C07275=1014.277,-66.718,394.005,165.149,59.305,160.508
C07276=1014.282,-66.468,393.994,165.151,59.299,160.507
C07277=1014.287,-66.219,393.985,165.154,59.292,160.507
C07278=1014.291,-65.969,393.976,165.157,59.286,160.507
C07279=1014.296,-65.719,393.966,165.160,59.279,160.506
C07280=1014.301,-65.470,393.956,165.161,59.272,160.505
C07281=1014.306,-65.219,393.947,165.165,59.265,160.505
C07282=1014.311,-64.970,393.937,165.167,59.258,160.504
C07283=1014.316,-64.720,393.927,165.170,59.251,160.504
C07284=1014.320,-64.470,393.918,165.173,59.245,160.503
C07285=1014.325,-64.221,393.908,165.175,59.238,160.502
C07286=1014.331,-63.971,393.898,165.177,59.231,160.502
C07287=1014.335,-63.721,393.889,165.180,59.223,160.501
C07288=1014.340,-63.472,393.879,165.183,59.217,160.501
C07289=1014.345,-63.222,393.869,165.186,59.210,160.500
C07290=1014.350,-62.972,393.859,165.187,59.203,160.500
C07291=1014.355,-62.722,393.850,165.190,59.196,160.499
C07292=1014.360,-62.473,393.840,165.193,59.189,160.498
C07293=1014.364,-62.223,393.830,165.196,59.182,160.498
C07294=1014.370,-61.973,393.820,165.199,59.175,160.497
C07295=1014.374,-61.723,393.811,165.201,59.168,160.497
C07296=1014.379,-61.474,393.801,165.203,59.161,160.496
C07297=1014.384,-61.224,393.792,165.205,59.154,160.495
C07298=1014.390,-60.974,393.781,165.208,59.147,160.495
C07299=1014.394,-60.724,393.772,165.211,59.140,160.494
C07300=1014.399,-60.475,393.763,165.214,59.133,160.494
C07301=1014.404,-60.225,393.752,165.217,59.126,160.493
C07302=1014.409,-59.975,393.743,165.219,59.119,160.493
C07303=1014.413,-59.725,393.732,165.222,59.112,160.492
C07304=1014.418,-59.475,393.723,165.225,59.104,160.492
C07305=1014.423,-59.225,393.713,165.227,59.097,160.491
C07306=1014.428,-58.976,393.703,165.229,59.091,160.490
C07307=1014.433,-58.726,393.693,165.231,59.083,160.489
C07308=1014.438,-58.476,393.683,165.234,59.076,160.489
C07309=1014.443,-58.227,393.673,165.237,59.069,160.488
C07310=1014.449,-57.977,393.663,165.239,59.062,160.488
C07311=1014.453,-57.727,393.654,165.242,59.055,160.487
C07312=1014.458,-57.477,393.644,165.245,59.048,160.486
C07313=1014.463,-57.227,393.634,165.247,59.040,160.486
C07314=1014.468,-56.978,393.624,165.250,59.033,160.485
C07315=1014.474,-56.728,393.614,165.253,59.026,160.485
C07316=1014.478,-56.478,393.604,165.255,59.018,160.484
C07317=1014.483,-56.229,393.595,165.257,59.011,160.483
C07318=1014.489,-55.979,393.584,165.260,59.004,160.483
C07319=1014.494,-55.729,393.575,165.263,58.997,160.482
C07320=1014.498,-55.480,393.565,165.265,58.989,160.481
C07321=1014.504,-55.229,393.555,165.268,58.982,160.481
C07322=1014.508,-54.980,393.546,165.271,58.975,160.480
C07323=1014.514,-54.730,393.535,165.273,58.967,160.479
C07324=1014.519,-54.480,393.526,165.275,58.960,160.479
C07325=1014.524,-54.204,393.514,165.278,58.952,160.478
C07326=1014.530,-53.930,393.503,165.282,58.944,160.477
C07327=1014.535,-53.653,393.492,165.284,58.936,160.477
C07328=1014.541,-53.378,393.481,165.287,58.928,160.476
C07329=1014.546,-53.128,393.471,165.290,58.921,160.475
C07330=1014.551,-52.879,393.461,165.292,58.913,160.474
C07331=1014.556,-52.629,393.451,165.295,58.906,160.474
C07332=1014.561,-52.379,393.441,165.298,58.898,160.473
C07333=1014.566,-52.130,393.432,165.300,58.890,160.472
C07334=1014.572,-51.880,393.421,165.303,58.883,160.472
C07335=1014.576,-51.630,393.412,165.306,58.876,160.471
C07336=1014.581,-51.380,393.401,165.308,58.868,160.470
C07337=1014.586,-51.130,393.391,165.310,58.861,160.470
C07338=1014.591,-50.880,393.381,165.313,58.854,160.469
C07339=1014.596,-50.631,393.369,165.316,58.847,160.468
C07340=1014.601,-50.381,393.360,165.318,58.839,160.468
C07341=1014.606,-50.131,393.349,165.321,58.832,160.467
C07342=1014.611,-49.881,393.339,165.324,58.825,160.467
C07343=1014.616,-49.632,393.328,165.326,58.818,160.466
C07344=1014.621,-49.382,393.318,165.329,58.811,160.465
C07345=1014.625,-49.132,393.307,165.331,58.803,160.464
C07346=1014.630,-48.883,393.297,165.334,58.796,160.464
C07347=1014.636,-48.633,393.286,165.337,58.789,160.463
C07348=1014.640,-48.383,393.276,165.339,58.782,160.463
C07349=1014.646,-48.134,393.265,165.342,58.774,160.462
C07350=1014.650,-47.883,393.254,165.345,58.767,160.461
C07351=1014.655,-47.634,393.245,165.347,58.759,160.461
C07352=1014.660,-47.384,393.233,165.349,58.752,160.460
C07353=1014.665,-47.135,393.223,165.352,58.745,160.459
C07354=1014.670,-46.884,393.213,165.355,58.738,160.459
C07355=1014.675,-46.635,393.202,165.357,58.730,160.458
C07356=1014.680,-46.385,393.191,165.359,58.723,160.457
C07357=1014.685,-46.135,393.180,165.362,58.716,160.457
C07358=1014.689,-45.886,393.170,165.365,58.709,160.456
C07359=1014.695,-45.636,393.160,165.367,58.701,160.455
C07360=1014.699,-45.386,393.149,165.370,58.694,160.454
C07361=1014.705,-45.136,393.139,165.372,58.687,160.454
C07362=1014.710,-44.887,393.128,165.374,58.679,160.453
C07363=1014.714,-44.637,393.117,165.377,58.672,160.452
C07364=1014.720,-44.388,393.106,165.380,58.664,160.452
C07365=1014.725,-44.137,393.096,165.383,58.656,160.451
C07366=1014.730,-43.888,393.086,165.386,58.649,160.450
C07367=1014.735,-43.638,393.074,165.388,58.642,160.450
C07368=1014.740,-43.389,393.065,165.390,58.634,160.449
C07369=1014.745,-43.139,393.053,165.393,58.627,160.448
C07370=1014.750,-42.889,393.043,165.395,58.619,160.447
C07371=1014.754,-42.640,393.032,165.398,58.612,160.447
C07372=1014.760,-42.390,393.022,165.400,58.604,160.446
C07373=1014.765,-42.140,393.010,165.404,58.596,160.445
C07374=1014.770,-41.890,393.000,165.406,58.589,160.445
C07375=1014.775,-41.641,392.989,165.409,58.582,160.444
C07376=1014.780,-41.390,392.979,165.411,58.574,160.443
C07377=1014.785,-41.141,392.967,165.413,58.567,160.442
C07378=1014.790,-40.891,392.958,165.416,58.559,160.442
C07379=1014.795,-40.641,392.946,165.419,58.551,160.441
C07380=1014.800,-40.391,392.936,165.421,58.543,160.440
C07381=1014.806,-40.143,392.925,165.424,58.536,160.440
C07382=1014.811,-39.893,392.914,165.426,58.528,160.439
C07383=1014.816,-39.643,392.904,165.429,58.521,160.438
C07384=1014.821,-39.393,392.892,165.431,58.513,160.437
C07385=1014.825,-39.143,392.882,165.434,58.506,160.437
C07386=1014.830,-38.893,392.870,165.438,58.499,160.436
C07387=1014.836,-38.644,392.860,165.440,58.491,160.435
C07388=1014.840,-38.395,392.848,165.442,58.484,160.435
C07389=1014.846,-38.119,392.837,165.445,58.476,160.434
C07390=1014.852,-37.844,392.824,165.448,58.468,160.433
C07391=1014.857,-37.568,392.812,165.450,58.459,160.432
C07392=1014.862,-37.293,392.800,165.453,58.450,160.431
C07393=1014.867,-37.043,392.789,165.456,58.443,160.431
C07394=1014.872,-36.793,392.777,165.458,58.435,160.430
C07395=1014.877,-36.544,392.766,165.461,58.428,160.429
C07396=1014.882,-36.295,392.755,165.463,58.420,160.428
C07397=1014.887,-36.044,392.745,165.466,58.413,160.428
C07398=1014.892,-35.795,392.733,165.468,58.405,160.427
C07399=1014.897,-35.545,392.722,165.472,58.398,160.426
C07400=1014.902,-35.295,392.710,165.474,58.390,160.425
C07401=1014.907,-35.046,392.700,165.477,58.383,160.425
C07402=1014.912,-34.796,392.689,165.479,58.375,160.424
C07403=1014.917,-34.546,392.678,165.481,58.367,160.423
C07404=1014.922,-34.296,392.666,165.484,58.360,160.422
C07405=1014.928,-34.047,392.655,165.487,58.352,160.422
C07406=1014.932,-33.798,392.644,165.490,58.345,160.421
C07407=1014.937,-33.548,392.633,165.492,58.337,160.420
C07408=1014.942,-33.298,392.621,165.494,58.329,160.419
C07409=1014.948,-33.048,392.611,165.497,58.322,160.419
C07410=1014.953,-32.798,392.600,165.500,58.314,160.418
C07411=1014.958,-32.548,392.588,165.502,58.306,160.417
C07412=1014.963,-32.299,392.577,165.505,58.299,160.417
C07413=1014.967,-32.049,392.565,165.507,58.291,160.416
C07414=1014.973,-31.800,392.555,165.510,58.283,160.415
C07415=1014.978,-31.550,392.543,165.512,58.275,160.414
C07416=1014.983,-31.300,392.532,165.515,58.268,160.413
C07417=1014.988,-31.051,392.520,165.517,58.260,160.412
C07418=1014.994,-30.801,392.509,165.519,58.252,160.412
C07419=1014.998,-30.551,392.499,165.523,58.245,160.411
C07420=1015.003,-30.301,392.487,165.525,58.237,160.410
C07421=1015.008,-30.051,392.476,165.527,58.229,160.409
C07422=1015.013,-29.802,392.465,165.531,58.221,160.409
C07423=1015.018,-29.552,392.454,165.533,58.213,160.408
C07424=1015.023,-29.303,392.442,165.536,58.206,160.407
C07425=1015.028,-29.053,392.431,165.538,58.198,160.406
C07426=1015.033,-28.803,392.419,165.541,58.190,160.406
C07427=1015.039,-28.554,392.408,165.543,58.182,160.405
C07428=1015.044,-28.304,392.397,165.545,58.174,160.404
C07429=1015.049,-28.054,392.385,165.548,58.166,160.403
C07430=1015.054,-27.804,392.374,165.551,58.158,160.402
C07431=1015.059,-27.554,392.362,165.553,58.151,160.401
C07432=1015.064,-27.305,392.351,165.556,58.143,160.401
C07433=1015.069,-27.055,392.339,165.558,58.136,160.400
C07434=1015.074,-26.806,392.327,165.562,58.128,160.399
C07435=1015.079,-26.556,392.316,165.564,58.120,160.398
C07436=1015.084,-26.306,392.304,165.566,58.113,160.397
C07437=1015.089,-26.056,392.293,165.568,58.105,160.397
C07438=1015.095,-25.807,392.281,165.571,58.098,160.396
C07439=1015.100,-25.557,392.269,165.574,58.089,160.395
C07440=1015.105,-25.307,392.258,165.576,58.082,160.394
C07441=1015.110,-25.058,392.246,165.579,58.074,160.393
C07442=1015.115,-24.808,392.235,165.581,58.067,160.393
C07443=1015.120,-24.559,392.223,165.585,58.059,160.392
C07444=1015.124,-24.308,392.211,165.587,58.051,160.391
C07445=1015.129,-24.059,392.199,165.589,58.043,160.390
C07446=1015.134,-23.809,392.188,165.591,58.035,160.389
C07447=1015.140,-23.560,392.175,165.595,58.028,160.389
C07448=1015.145,-23.310,392.164,165.597,58.020,160.388
C07449=1015.150,-23.060,392.152,165.599,58.012,160.387
C07450=1015.155,-22.811,392.140,165.602,58.004,160.386
C07451=1015.160,-22.561,392.129,165.605,57.996,160.386
C07452=1015.165,-22.311,392.117,165.607,57.988,160.385
C07453=1015.171,-22.035,392.104,165.610,57.979,160.384
C07454=1015.176,-21.758,392.091,165.613,57.971,160.383
C07455=1015.182,-21.483,392.079,165.616,57.962,160.382
C07456=1015.188,-21.207,392.065,165.618,57.953,160.381
C07457=1015.193,-20.957,392.054,165.621,57.946,160.380
C07458=1015.198,-20.707,392.042,165.623,57.938,160.380
C07459=1015.204,-20.457,392.030,165.627,57.930,160.379
C07460=1015.208,-20.207,392.018,165.629,57.922,160.378
C07461=1015.213,-19.957,392.006,165.631,57.915,160.377
C07462=1015.218,-19.708,391.994,165.634,57.906,160.376
C07463=1015.223,-19.458,391.983,165.636,57.899,160.375
C07464=1015.228,-19.209,391.970,165.639,57.891,160.375
C07465=1015.233,-18.959,391.959,165.642,57.883,160.374
C07466=1015.238,-18.709,391.947,165.643,57.874,160.373
C07467=1015.244,-18.460,391.935,165.646,57.866,160.372
C07468=1015.249,-18.210,391.924,165.649,57.858,160.371
C07469=1015.255,-17.961,391.911,165.651,57.850,160.370
C07470=1015.260,-17.711,391.900,165.653,57.843,160.369
C07471=1015.265,-17.461,391.888,165.657,57.834,160.369
C07472=1015.270,-17.212,391.876,165.659,57.827,160.368
C07473=1015.275,-16.962,391.865,165.662,57.818,160.367
C07474=1015.280,-16.712,391.852,165.664,57.811,160.366
C07475=1015.285,-16.462,391.840,165.667,57.803,160.365
C07476=1015.290,-16.212,391.829,165.669,57.794,160.364
C07477=1015.295,-15.963,391.816,165.672,57.786,160.363
C07478=1015.301,-15.714,391.804,165.674,57.778,160.362
C07479=1015.305,-15.464,391.792,165.677,57.770,160.362
C07480=1015.311,-15.214,391.780,165.680,57.763,160.361
C07481=1015.316,-14.964,391.768,165.682,57.756,160.360
C07482=1015.320,-14.714,391.755,165.684,57.748,160.359
C07483=1015.326,-14.465,391.743,165.688,57.740,160.359
C07484=1015.330,-14.215,391.731,165.690,57.732,160.358
C07485=1015.336,-13.965,391.719,165.692,57.723,160.356
C07486=1015.341,-13.715,391.707,165.695,57.715,160.356
C07487=1015.346,-13.466,391.694,165.697,57.707,160.355
C07488=1015.351,-13.217,391.682,165.699,57.700,160.354
C07489=1015.356,-12.967,391.671,165.703,57.691,160.353
C07490=1015.361,-12.717,391.657,165.705,57.684,160.352
C07491=1015.366,-12.468,391.645,165.707,57.676,160.351
C07492=1015.372,-12.218,391.633,165.709,57.668,160.351
C07493=1015.376,-11.968,391.621,165.713,57.660,160.350
C07494=1015.382,-11.718,391.608,165.715,57.652,160.349
C07495=1015.387,-11.469,391.596,165.717,57.645,160.348
C07496=1015.391,-11.219,391.584,165.721,57.636,160.347
C07497=1015.397,-10.970,391.572,165.722,57.628,160.346
C07498=1015.403,-10.720,391.559,165.726,57.620,160.345
C07499=1015.407,-10.471,391.547,165.728,57.612,160.345
C07500=1015.412,-10.221,391.535,165.730,57.604,160.344
C07501=1015.417,-9.971,391.522,165.733,57.596,160.343
C07502=1015.423,-9.721,391.510,165.735,57.588,160.342
C07503=1015.428,-9.472,391.498,165.737,57.580,160.341
C07504=1015.432,-9.222,391.486,165.741,57.572,160.340
C07505=1015.438,-8.972,391.473,165.743,57.564,160.339
C07506=1015.443,-8.723,391.461,165.745,57.556,160.338
C07507=1015.448,-8.474,391.448,165.748,57.547,160.337
C07508=1015.453,-8.224,391.437,165.750,57.540,160.337
C07509=1015.460,-7.880,391.420,165.754,57.528,160.335
C07510=1015.468,-7.536,391.402,165.758,57.517,160.334
C07511=1015.475,-7.193,391.385,165.761,57.506,160.333
C07512=1015.482,-6.850,391.368,165.765,57.495,160.332
C07513=1015.486,-6.632,391.358,165.767,57.488,160.331
C07514=1015.491,-6.415,391.346,165.769,57.480,160.330
C07515=1015.496,-6.199,391.335,165.771,57.474,160.329
C07516=1015.500,-5.982,391.324,165.773,57.466,160.328
C07517=1015.505,-5.765,391.314,165.775,57.460,160.328
C07518=1015.509,-5.548,391.303,165.778,57.453,160.327
C07519=1015.514,-5.331,391.292,165.780,57.445,160.326
C07520=1015.518,-5.114,391.281,165.782,57.438,160.325
C07521=1015.523,-4.865,391.270,165.785,57.430,160.325
C07522=1015.528,-4.614,391.257,165.787,57.422,160.323
C07523=1015.534,-4.365,391.245,165.790,57.414,160.323
C07524=1015.539,-4.115,391.231,165.793,57.406,160.322
C07525=1015.543,-3.866,391.219,165.795,57.398,160.321
C07526=1015.548,-3.616,391.206,165.797,57.390,160.320
C07527=1015.554,-3.367,391.193,165.800,57.382,160.319
C07528=1015.559,-3.117,391.180,165.802,57.374,160.318
C07529=1015.564,-2.867,391.167,165.805,57.366,160.317
C07530=1015.568,-2.618,391.154,165.808,57.358,160.317
C07531=1015.574,-2.368,391.142,165.810,57.350,160.316
C07532=1015.579,-2.118,391.129,165.812,57.342,160.315
C07533=1015.583,-1.869,391.116,165.815,57.334,160.314
C07534=1015.589,-1.619,391.103,165.818,57.326,160.313
C07535=1015.594,-1.370,391.090,165.820,57.318,160.312
C07536=1015.599,-1.120,391.077,165.822,57.310,160.311
C07537=1015.604,-0.870,391.064,165.825,57.302,160.310
C07538=1015.609,-0.621,391.052,165.828,57.294,160.309
C07539=1015.614,-0.371,391.038,165.830,57.286,160.308
C07540=1015.619,-0.121,391.026,165.833,57.277,160.307
C07541=1015.624,0.129,391.013,165.835,57.270,160.307
C07542=1015.630,0.377,391.000,165.838,57.262,160.306
C07543=1015.635,0.628,390.986,165.840,57.253,160.305
C07544=1015.639,0.877,390.974,165.842,57.245,160.304
C07545=1015.644,1.127,390.961,165.846,57.237,160.303
C07546=1015.650,1.376,390.948,165.848,57.229,160.302
C07547=1015.655,1.625,390.935,165.850,57.221,160.301
C07548=1015.660,1.875,390.922,165.853,57.213,160.300
C07549=1015.665,2.125,390.909,165.855,57.205,160.299
C07550=1015.670,2.375,390.896,165.857,57.197,160.298
C07551=1015.675,2.624,390.883,165.861,57.189,160.298
C07552=1015.681,2.874,390.870,165.862,57.180,160.296
C07553=1015.685,3.123,390.857,165.866,57.172,160.296
C07554=1015.691,3.373,390.844,165.868,57.164,160.295
C07555=1015.696,3.622,390.831,165.870,57.156,160.294
C07556=1015.701,3.872,390.818,165.873,57.148,160.293
C07557=1015.706,4.122,390.805,165.875,57.140,160.292
C07558=1015.712,4.372,390.792,165.879,57.132,160.291
C07559=1015.716,4.621,390.779,165.880,57.123,160.290
C07560=1015.722,4.871,390.766,165.883,57.116,160.289
C07561=1015.726,5.120,390.753,165.886,57.107,160.288
C07562=1015.732,5.370,390.740,165.888,57.099,160.287
C07563=1015.738,5.620,390.727,165.891,57.090,160.286
C07564=1015.742,5.869,390.714,165.893,57.083,160.285
C07565=1015.748,6.119,390.700,165.896,57.074,160.284
C07566=1015.753,6.368,390.688,165.898,57.066,160.284
C07567=1015.758,6.618,390.675,165.901,57.057,160.283
C07568=1015.763,6.867,390.661,165.903,57.050,160.282
C07569=1015.768,7.117,390.648,165.905,57.041,160.280
C07570=1015.774,7.367,390.635,165.909,57.033,160.280
C07571=1015.779,7.616,390.622,165.910,57.025,160.279
C07572=1015.784,7.866,390.609,165.913,57.016,160.278
C07573=1015.789,8.116,390.596,165.916,57.008,160.277
C07574=1015.795,8.365,390.583,165.919,56.999,160.276
C07575=1015.799,8.614,390.570,165.921,56.992,160.275
C07576=1015.805,8.865,390.557,165.924,56.983,160.274
C07577=1015.810,9.114,390.543,165.926,56.974,160.273
C07578=1015.815,9.363,390.531,165.929,56.966,160.272
C07579=1015.821,9.613,390.517,165.931,56.958,160.271
C07580=1015.825,9.862,390.504,165.934,56.949,160.270
C07581=1015.832,10.143,390.489,165.936,56.940,160.269
C07582=1015.837,10.423,390.474,165.939,56.931,160.268
C07583=1015.843,10.704,390.459,165.943,56.922,160.267
C07584=1015.849,10.984,390.445,165.945,56.912,160.266
C07585=1015.855,11.233,390.431,165.947,56.904,160.264
C07586=1015.860,11.483,390.419,165.950,56.896,160.264
C07587=1015.865,11.732,390.405,165.952,56.887,160.263
C07588=1015.870,11.982,390.392,165.955,56.878,160.262
C07589=1015.876,12.231,390.379,165.958,56.870,160.261
C07590=1015.881,12.481,390.366,165.960,56.862,160.260
C07591=1015.887,12.731,390.352,165.963,56.853,160.259
C07592=1015.891,12.980,390.339,165.965,56.845,160.258
C07593=1015.897,13.230,390.325,165.968,56.836,160.257
C07594=1015.902,13.480,390.312,165.970,56.828,160.256
C07595=1015.907,13.730,390.298,165.972,56.820,160.255
C07596=1015.912,13.979,390.285,165.976,56.812,160.254
C07597=1015.917,14.229,390.271,165.977,56.804,160.253
C07598=1015.923,14.478,390.258,165.981,56.795,160.252
C07599=1015.927,14.728,390.245,165.983,56.787,160.251
C07600=1015.933,14.977,390.231,165.986,56.778,160.250
C07601=1015.938,15.227,390.217,165.988,56.771,160.249
C07602=1015.943,15.476,390.204,165.990,56.762,160.248
C07603=1015.948,15.726,390.190,165.993,56.754,160.247
C07604=1015.954,15.976,390.177,165.995,56.746,160.246
C07605=1015.959,16.225,390.163,165.998,56.737,160.245
C07606=1015.963,16.475,390.149,166.000,56.729,160.244
C07607=1015.969,16.724,390.135,166.003,56.721,160.243
C07608=1015.974,16.974,390.122,166.005,56.712,160.242
C07609=1015.979,17.224,390.109,166.008,56.704,160.241
C07610=1015.984,17.473,390.095,166.011,56.696,160.240
C07611=1015.990,17.723,390.081,166.012,56.688,160.239
C07612=1015.995,17.972,390.067,166.015,56.679,160.238
C07613=1016.000,18.222,390.054,166.018,56.671,160.237
C07614=1016.005,18.471,390.041,166.021,56.662,160.236
C07615=1016.011,18.721,390.027,166.023,56.654,160.235
C07616=1016.016,18.970,390.013,166.025,56.645,160.234
C07617=1016.022,19.220,389.999,166.028,56.638,160.233
C07618=1016.025,19.470,389.986,166.031,56.629,160.232
C07619=1016.031,19.719,389.972,166.033,56.621,160.232
C07620=1016.036,19.969,389.958,166.035,56.613,160.230
C07621=1016.042,20.219,389.944,166.038,56.604,160.229
C07622=1016.047,20.467,389.930,166.040,56.596,160.228
C07623=1016.051,20.717,389.916,166.043,56.588,160.228
C07624=1016.057,20.967,389.902,166.045,56.579,160.226
C07625=1016.062,21.216,389.888,166.048,56.571,160.225
C07626=1016.068,21.467,389.875,166.051,56.563,160.225
C07627=1016.072,21.716,389.861,166.054,56.554,160.224
C07628=1016.077,21.965,389.847,166.056,56.546,160.222
C07629=1016.083,22.215,389.833,166.057,56.538,160.221
C07630=1016.088,22.465,389.819,166.061,56.530,160.221
C07631=1016.094,22.714,389.806,166.063,56.521,160.219
C07632=1016.098,22.963,389.791,166.066,56.513,160.219
C07633=1016.103,23.213,389.778,166.068,56.504,160.217
C07634=1016.109,23.463,389.764,166.071,56.496,160.217
C07635=1016.114,23.712,389.750,166.073,56.488,160.216
C07636=1016.120,23.962,389.736,166.076,56.479,160.215
C07637=1016.124,24.212,389.722,166.078,56.471,160.213
C07638=1016.130,24.461,389.708,166.081,56.462,160.212
C07639=1016.135,24.710,389.694,166.083,56.454,160.212
C07640=1016.140,24.960,389.680,166.086,56.446,160.211
C07641=1016.145,25.209,389.666,166.088,56.437,160.210
C07642=1016.150,25.459,389.652,166.091,56.429,160.209
C07643=1016.156,25.709,389.638,166.093,56.420,160.207
C07644=1016.161,25.958,389.624,166.096,56.412,160.206
C07645=1016.167,26.240,389.609,166.099,56.403,160.205
C07646=1016.173,26.521,389.593,166.102,56.393,160.204
C07647=1016.179,26.803,389.577,166.105,56.383,160.203
C07648=1016.184,27.085,389.561,166.107,56.374,160.202
C07649=1016.189,27.335,389.547,166.109,56.366,160.201
C07650=1016.195,27.584,389.532,166.112,56.357,160.200
C07651=1016.200,27.834,389.518,166.115,56.349,160.199
C07652=1016.205,28.083,389.504,166.118,56.341,160.198
C07653=1016.210,28.333,389.490,166.120,56.332,160.197
C07654=1016.216,28.583,389.476,166.122,56.324,160.196
C07655=1016.220,28.832,389.462,166.125,56.316,160.195
C07656=1016.225,29.081,389.447,166.127,56.308,160.194
C07657=1016.230,29.331,389.433,166.130,56.299,160.193
C07658=1016.236,29.580,389.419,166.132,56.291,160.192
C07659=1016.241,29.830,389.405,166.135,56.282,160.191
C07660=1016.246,30.080,389.390,166.138,56.274,160.190
C07661=1016.252,30.329,389.376,166.140,56.266,160.189
C07662=1016.256,30.579,389.361,166.143,56.257,160.188
C07663=1016.262,30.828,389.348,166.144,56.249,160.187
C07664=1016.267,31.078,389.333,166.147,56.240,160.186
C07665=1016.272,31.327,389.319,166.149,56.232,160.185
C07666=1016.277,31.577,389.304,166.152,56.223,160.184
C07667=1016.283,31.827,389.290,166.155,56.216,160.183
C07668=1016.287,32.076,389.276,166.158,56.207,160.182
C07669=1016.293,32.325,389.261,166.160,56.199,160.181
C07670=1016.298,32.575,389.247,166.163,56.190,160.180
C07671=1016.303,32.825,389.233,166.165,56.182,160.179
C07672=1016.308,33.074,389.218,166.168,56.173,160.178
C07673=1016.314,33.324,389.204,166.170,56.165,160.177
C07674=1016.319,33.574,389.189,166.173,56.156,160.176
C07675=1016.324,33.823,389.175,166.175,56.148,160.174
C07676=1016.329,34.072,389.160,166.178,56.139,160.174
C07677=1016.335,34.322,389.146,166.180,56.131,160.172
C07678=1016.339,34.572,389.132,166.183,56.122,160.171
C07679=1016.345,34.821,389.117,166.185,56.115,160.171
C07680=1016.351,35.070,389.104,166.188,56.106,160.170
C07681=1016.355,35.320,389.089,166.190,56.098,160.169
C07682=1016.361,35.569,389.075,166.193,56.089,160.168
C07683=1016.366,35.819,389.060,166.195,56.081,160.166
C07684=1016.372,36.068,389.045,166.198,56.072,160.165
C07685=1016.376,36.318,389.031,166.200,56.064,160.164
C07686=1016.381,36.568,389.017,166.204,56.055,160.163
C07687=1016.387,36.817,389.002,166.206,56.047,160.162
C07688=1016.392,37.067,388.988,166.207,56.039,160.161
C07689=1016.397,37.316,388.972,166.211,56.030,160.160
C07690=1016.401,37.566,388.958,166.213,56.022,160.159
C07691=1016.407,37.815,388.943,166.216,56.013,160.158
C07692=1016.412,38.065,388.929,166.218,56.005,160.157
C07693=1016.417,38.314,388.914,166.221,55.997,160.156
C07694=1016.422,38.564,388.900,166.223,55.988,160.155
C07695=1016.427,38.813,388.885,166.225,55.980,160.154
C07696=1016.433,39.063,388.869,166.228,55.972,160.153
C07697=1016.438,39.313,388.855,166.230,55.963,160.152
C07698=1016.444,39.562,388.840,166.233,55.955,160.151
C07699=1016.448,39.812,388.826,166.235,55.946,160.150
C07700=1016.453,40.061,388.810,166.238,55.938,160.149
C07701=1016.458,40.311,388.796,166.240,55.929,160.148
C07702=1016.464,40.560,388.781,166.243,55.921,160.147
C07703=1016.469,40.809,388.766,166.246,55.912,160.146
C07704=1016.474,41.059,388.752,166.248,55.904,160.145
C07705=1016.480,41.308,388.737,166.251,55.896,160.144
C07706=1016.484,41.558,388.723,166.253,55.887,160.143
C07707=1016.490,41.808,388.707,166.256,55.879,160.142
C07708=1016.495,42.057,388.692,166.258,55.870,160.140
C07709=1016.501,42.338,388.676,166.261,55.861,160.139
C07710=1016.507,42.620,388.659,166.264,55.852,160.138
C07711=1016.512,42.902,388.642,166.267,55.843,160.137
C07712=1016.518,43.184,388.625,166.270,55.833,160.136
C07713=1016.523,43.434,388.609,166.273,55.825,160.135
C07714=1016.528,43.683,388.595,166.275,55.816,160.134
C07715=1016.533,43.933,388.580,166.277,55.808,160.133
C07716=1016.538,44.182,388.565,166.280,55.800,160.132
C07717=1016.543,44.431,388.549,166.282,55.792,160.131
C07718=1016.548,44.680,388.534,166.284,55.784,160.130
C07719=1016.554,44.930,388.519,166.287,55.775,160.129
C07720=1016.558,45.180,388.504,166.290,55.767,160.128
C07721=1016.563,45.430,388.489,166.293,55.758,160.127
C07722=1016.568,45.679,388.474,166.295,55.750,160.126
C07723=1016.574,45.928,388.459,166.297,55.742,160.125
C07724=1016.579,46.177,388.443,166.300,55.734,160.124
C07725=1016.583,46.428,388.427,166.302,55.726,160.123
C07726=1016.589,46.677,388.412,166.304,55.717,160.122
C07727=1016.593,46.927,388.398,166.308,55.709,160.121
C07728=1016.598,47.176,388.383,166.310,55.701,160.120
C07729=1016.603,47.425,388.367,166.313,55.692,160.119
C07730=1016.608,47.675,388.352,166.315,55.684,160.118
C07731=1016.614,47.925,388.337,166.318,55.675,160.117
C07732=1016.619,48.174,388.321,166.320,55.667,160.116
C07733=1016.624,48.423,388.306,166.322,55.659,160.114
C07734=1016.629,48.672,388.291,166.325,55.650,160.114
C07735=1016.635,48.922,388.276,166.327,55.642,160.112
C07736=1016.640,49.172,388.261,166.330,55.633,160.111
C07737=1016.645,49.422,388.246,166.332,55.625,160.110
C07738=1016.650,49.671,388.231,166.336,55.616,160.109
C07739=1016.655,49.920,388.216,166.338,55.608,160.108
C07740=1016.660,50.170,388.200,166.340,55.600,160.107
C07741=1016.665,50.419,388.185,166.343,55.591,160.106
C07742=1016.670,50.669,388.170,166.345,55.583,160.105
C07743=1016.675,50.918,388.155,166.348,55.574,160.104
C07744=1016.681,51.168,388.139,166.350,55.566,160.103
C07745=1016.686,51.417,388.124,166.353,55.558,160.102
C07746=1016.691,51.666,388.109,166.355,55.549,160.101
C07747=1016.696,51.916,388.093,166.359,55.541,160.100
C07748=1016.702,52.166,388.078,166.361,55.533,160.099
C07749=1016.707,52.415,388.063,166.363,55.523,160.098
C07750=1016.712,52.664,388.048,166.365,55.515,160.097
C07751=1016.718,52.914,388.032,166.369,55.506,160.096
C07752=1016.722,53.164,388.016,166.371,55.498,160.095
C07753=1016.727,53.413,388.001,166.373,55.490,160.094
C07754=1016.732,53.662,387.986,166.376,55.481,160.093
C07755=1016.738,53.912,387.970,166.378,55.473,160.091
C07756=1016.743,54.161,387.955,166.381,55.465,160.091
C07757=1016.748,54.411,387.940,166.383,55.456,160.089
C07758=1016.753,54.661,387.924,166.386,55.447,160.088
C07759=1016.758,54.910,387.909,166.388,55.439,160.087
C07760=1016.763,55.159,387.894,166.391,55.430,160.086
C07761=1016.769,55.409,387.879,166.393,55.422,160.085
C07762=1016.774,55.658,387.863,166.397,55.414,160.084
C07763=1016.779,55.908,387.848,166.399,55.404,160.083
C07764=1016.785,56.158,387.833,166.401,55.396,160.082
C07765=1016.790,56.406,387.817,166.404,55.388,160.081
C07766=1016.795,56.656,387.802,166.407,55.379,160.080
C07767=1016.801,56.906,387.786,166.410,55.371,160.079
C07768=1016.806,57.155,387.771,166.411,55.362,160.077
C07769=1016.811,57.404,387.756,166.415,55.353,160.077
C07770=1016.817,57.654,387.740,166.417,55.345,160.075
C07771=1016.822,57.903,387.725,166.420,55.337,160.075
C07772=1016.826,58.153,387.709,166.422,55.328,160.073
C07773=1016.833,58.434,387.692,166.425,55.318,160.072
C07774=1016.839,58.716,387.675,166.428,55.309,160.071
C07775=1016.845,58.998,387.657,166.431,55.299,160.070
C07776=1016.850,59.280,387.640,166.434,55.289,160.068
C07777=1016.856,59.529,387.624,166.436,55.281,160.067
C07778=1016.861,59.778,387.609,166.439,55.272,160.066
C07779=1016.866,60.028,387.593,166.442,55.263,160.065
C07780=1016.872,60.278,387.578,166.444,55.255,160.064
C07781=1016.877,60.527,387.563,166.447,55.246,160.063
C07782=1016.882,60.777,387.547,166.449,55.237,160.062
C07783=1016.887,61.026,387.531,166.452,55.229,160.061
C07784=1016.892,61.275,387.515,166.454,55.221,160.060
C07785=1016.898,61.525,387.500,166.457,55.211,160.059
C07786=1016.903,61.774,387.485,166.460,55.203,160.058
C07787=1016.909,62.024,387.469,166.462,55.195,160.057
C07788=1016.914,62.273,387.453,166.465,55.185,160.055
C07789=1016.920,62.523,387.438,166.467,55.177,160.054
C07790=1016.925,62.772,387.423,166.470,55.169,160.053
C07791=1016.930,63.022,387.406,166.472,55.160,160.052
C07792=1016.935,63.271,387.391,166.476,55.152,160.051
C07793=1016.941,63.521,387.375,166.477,55.143,160.050
C07794=1016.945,63.770,387.359,166.481,55.135,160.049
C07795=1016.950,64.019,387.343,166.483,55.126,160.048
C07796=1016.956,64.269,387.328,166.486,55.118,160.047
C07797=1016.961,64.518,387.311,166.488,55.110,160.046
C07798=1016.966,64.768,387.296,166.491,55.100,160.045
C07799=1016.971,65.017,387.279,166.493,55.092,160.044
C07800=1016.976,65.267,387.264,166.496,55.084,160.043
C07801=1016.982,65.516,387.248,166.498,55.076,160.042
C07802=1016.987,65.766,387.232,166.502,55.067,160.041
C07803=1016.992,66.015,387.217,166.503,55.058,160.039
C07804=1016.997,66.265,387.200,166.507,55.050,160.038
C07805=1017.002,66.514,387.185,166.509,55.042,160.037
C07806=1017.008,66.763,387.168,166.512,55.033,160.036
C07807=1017.012,67.013,387.153,166.514,55.025,160.035
C07808=1017.018,67.262,387.136,166.516,55.016,160.034
C07809=1017.023,67.512,387.121,166.519,55.008,160.033
C07810=1017.028,67.761,387.104,166.521,54.999,160.032
C07811=1017.033,68.011,387.088,166.525,54.991,160.031
C07812=1017.039,68.260,387.072,166.527,54.983,160.030
C07813=1017.043,68.509,387.056,166.530,54.973,160.029
C07814=1017.049,68.759,387.040,166.532,54.965,160.028
C07815=1017.054,69.008,387.024,166.535,54.957,160.027
C07816=1017.059,69.258,387.008,166.537,54.949,160.026
C07817=1017.064,69.507,386.992,166.541,54.940,160.025
C07818=1017.070,69.756,386.975,166.543,54.932,160.024
C07819=1017.074,70.006,386.960,166.546,54.923,160.022
C07820=1017.079,70.256,386.943,166.548,54.915,160.021
C07821=1017.085,70.504,386.927,166.550,54.907,160.020
C07822=1017.090,70.755,386.911,166.553,54.898,160.019
C07823=1017.095,71.003,386.895,166.555,54.890,160.018
C07824=1017.100,71.253,386.878,166.558,54.881,160.017
C07825=1017.104,71.502,386.862,166.560,54.873,160.016
C07826=1017.110,71.752,386.846,166.564,54.864,160.015
C07827=1017.116,72.001,386.829,166.566,54.856,160.014
C07828=1017.121,72.251,386.814,166.569,54.848,160.013
C07829=1017.126,72.500,386.797,166.571,54.839,160.012
C07830=1017.130,72.749,386.781,166.574,54.830,160.011
C07831=1017.136,72.999,386.765,166.576,54.822,160.010
C07832=1017.141,73.248,386.749,166.580,54.814,160.009
C07833=1017.147,73.498,386.732,166.582,54.805,160.007
C07834=1017.152,73.747,386.716,166.585,54.796,160.006
C07835=1017.156,73.997,386.700,166.587,54.788,160.005
C07836=1017.162,74.246,386.683,166.590,54.780,160.004
C07837=1017.168,74.528,386.665,166.593,54.770,160.003
C07838=1017.174,74.809,386.647,166.595,54.761,160.002
C07839=1017.179,75.091,386.628,166.599,54.751,160.001
C07840=1017.185,75.373,386.609,166.602,54.741,159.999
C07841=1017.190,75.622,386.593,166.604,54.733,159.998
C07842=1017.196,75.871,386.577,166.607,54.724,159.997
C07843=1017.201,76.122,386.560,166.609,54.716,159.996
C07844=1017.206,76.370,386.545,166.612,54.707,159.995
C07845=1017.211,76.620,386.528,166.614,54.699,159.994
C07846=1017.216,76.870,386.511,166.618,54.691,159.993
C07847=1017.221,77.119,386.494,166.620,54.683,159.992
C07848=1017.227,77.368,386.478,166.623,54.673,159.991
C07849=1017.232,77.618,386.461,166.625,54.665,159.990
C07850=1017.237,77.867,386.445,166.627,54.657,159.989
C07851=1017.242,78.116,386.428,166.631,54.649,159.988
C07852=1017.247,78.365,386.411,166.633,54.641,159.987
C07853=1017.252,78.615,386.395,166.636,54.632,159.986
C07854=1017.257,78.865,386.378,166.638,54.623,159.984
C07855=1017.262,79.113,386.361,166.641,54.615,159.983
C07856=1017.267,79.363,386.344,166.644,54.607,159.982
C07857=1017.272,79.613,386.328,166.646,54.599,159.981
C07858=1017.277,79.862,386.311,166.649,54.590,159.980
C07859=1017.283,80.111,386.295,166.651,54.581,159.979
C07860=1017.288,80.361,386.278,166.654,54.573,159.978
C07861=1017.292,80.610,386.261,166.657,54.565,159.977
C07862=1017.298,80.859,386.245,166.660,54.557,159.976
C07863=1017.303,81.109,386.228,166.662,54.548,159.975
C07864=1017.307,81.358,386.211,166.665,54.539,159.974
C07865=1017.313,81.608,386.194,166.667,54.531,159.973
C07866=1017.318,81.857,386.178,166.670,54.523,159.972
C07867=1017.323,82.107,386.161,166.673,54.515,159.971
C07868=1017.328,82.356,386.144,166.675,54.506,159.969
C07869=1017.333,82.606,386.127,166.678,54.497,159.969
C07870=1017.339,82.855,386.111,166.681,54.489,159.968
C07871=1017.343,83.104,386.095,166.684,54.481,159.967
C07872=1017.349,83.354,386.078,166.686,54.472,159.965
C07873=1017.354,83.603,386.061,166.689,54.464,159.964
C07874=1017.359,83.853,386.044,166.691,54.456,159.963
C07875=1017.364,84.101,386.027,166.695,54.447,159.962
C07876=1017.369,84.351,386.010,166.697,54.438,159.961
C07877=1017.374,84.601,385.993,166.700,54.430,159.960
C07878=1017.379,84.850,385.977,166.702,54.422,159.959
C07879=1017.384,85.099,385.960,166.705,54.413,159.958
C07880=1017.389,85.349,385.943,166.707,54.405,159.957
C07881=1017.395,85.598,385.926,166.711,54.396,159.956
C07882=1017.401,85.848,385.910,166.713,54.388,159.955
C07883=1017.406,86.096,385.893,166.716,54.379,159.954
C07884=1017.411,86.346,385.876,166.718,54.371,159.953
C07885=1017.416,86.595,385.859,166.721,54.362,159.951
C07886=1017.421,86.845,385.842,166.724,54.354,159.950
C07887=1017.426,87.094,385.826,166.727,54.346,159.949
C07888=1017.431,87.344,385.809,166.729,54.337,159.948
C07889=1017.436,87.593,385.791,166.732,54.328,159.947
C07890=1017.442,87.842,385.774,166.734,54.320,159.946
C07891=1017.447,88.092,385.758,166.737,54.311,159.945
C07892=1017.452,88.341,385.741,166.740,54.303,159.944
C07893=1017.457,88.591,385.724,166.743,54.294,159.943
C07894=1017.462,88.840,385.707,166.746,54.286,159.942
C07895=1017.467,89.089,385.690,166.748,54.278,159.941
C07896=1017.473,89.339,385.673,166.751,54.270,159.940
C07897=1017.478,89.588,385.655,166.754,54.260,159.938
C07898=1017.483,89.837,385.639,166.756,54.252,159.937
C07899=1017.487,90.087,385.621,166.759,54.244,159.937
C07900=1017.493,90.336,385.604,166.762,54.236,159.935
C07901=1017.499,90.618,385.585,166.765,54.227,159.934
C07902=1017.504,90.899,385.565,166.768,54.217,159.933
C07903=1017.510,91.182,385.546,166.771,54.208,159.932
C07904=1017.515,91.463,385.527,166.774,54.198,159.931
C07905=1017.521,91.712,385.509,166.777,54.189,159.930
C07906=1017.525,91.962,385.492,166.779,54.181,159.928
C07907=1017.531,92.211,385.474,166.783,54.173,159.928
C07908=1017.536,92.461,385.457,166.785,54.165,159.926
C07909=1017.542,92.710,385.440,166.788,54.156,159.925
C07910=1017.546,92.960,385.422,166.790,54.148,159.924
C07911=1017.551,93.209,385.406,166.793,54.140,159.923
C07912=1017.556,93.458,385.388,166.796,54.131,159.922
C07913=1017.562,93.707,385.371,166.798,54.123,159.921
C07914=1017.566,93.957,385.353,166.801,54.114,159.920
C07915=1017.572,94.207,385.336,166.804,54.106,159.919
C07916=1017.577,94.456,385.319,166.807,54.097,159.918
C07917=1017.582,94.705,385.302,166.809,54.089,159.917
C07918=1017.587,94.955,385.284,166.812,54.081,159.916
C07919=1017.592,95.204,385.267,166.814,54.072,159.915
C07920=1017.597,95.453,385.250,166.818,54.064,159.914
C07921=1017.602,95.702,385.233,166.820,54.056,159.913
C07922=1017.607,95.952,385.215,166.824,54.047,159.912
C07923=1017.612,96.201,385.198,166.826,54.039,159.910
C07924=1017.618,96.450,385.180,166.829,54.030,159.909
C07925=1017.623,96.699,385.163,166.831,54.022,159.908
C07926=1017.628,96.949,385.145,166.834,54.013,159.907
C07927=1017.633,97.198,385.128,166.837,54.005,159.906
C07928=1017.639,97.448,385.111,166.840,53.996,159.905
C07929=1017.644,97.697,385.093,166.842,53.988,159.904
C07930=1017.649,97.947,385.076,166.846,53.980,159.903
C07931=1017.654,98.195,385.059,166.847,53.971,159.902
C07932=1017.659,98.444,385.041,166.851,53.963,159.901
C07933=1017.664,98.694,385.024,166.854,53.954,159.900
C07934=1017.669,98.943,385.006,166.856,53.946,159.899
C07935=1017.674,99.193,384.989,166.860,53.937,159.898
C07936=1017.680,99.442,384.972,166.862,53.929,159.897
C07937=1017.685,99.691,384.953,166.865,53.921,159.896
C07938=1017.689,99.941,384.935,166.868,53.912,159.894
C07939=1017.695,100.190,384.918,166.870,53.904,159.893
C07940=1017.699,100.440,384.900,166.873,53.896,159.892
C07941=1017.705,100.689,384.883,166.876,53.888,159.891
C07942=1017.710,100.938,384.865,166.879,53.879,159.890
C07943=1017.715,101.188,384.848,166.881,53.871,159.889
C07944=1017.720,101.437,384.830,166.885,53.862,159.888
C07945=1017.725,101.686,384.812,166.887,53.855,159.887
C07946=1017.730,101.936,384.794,166.889,53.846,159.886
C07947=1017.735,102.185,384.776,166.893,53.838,159.885
C07948=1017.740,102.435,384.759,166.895,53.830,159.884
C07949=1017.745,102.684,384.741,166.899,53.821,159.883
C07950=1017.750,102.933,384.723,166.900,53.813,159.882
C07951=1017.755,103.182,384.705,166.904,53.804,159.881
C07952=1017.760,103.431,384.687,166.906,53.796,159.880
C07953=1017.765,103.681,384.669,166.910,53.788,159.879
C07954=1017.771,103.930,384.652,166.912,53.779,159.878
C07955=1017.775,104.180,384.634,166.915,53.771,159.877
C07956=1017.781,104.429,384.617,166.918,53.763,159.876
C07957=1017.786,104.678,384.598,166.921,53.754,159.874
C07958=1017.791,104.927,384.581,166.923,53.746,159.873
C07959=1017.796,105.177,384.563,166.927,53.738,159.873
C07960=1017.801,105.426,384.545,166.929,53.730,159.871
C07961=1017.806,105.675,384.527,166.932,53.721,159.870
C07962=1017.811,105.924,384.509,166.935,53.713,159.869
C07963=1017.816,106.174,384.492,166.938,53.704,159.868
C07964=1017.821,106.423,384.474,166.940,53.696,159.867
C07965=1017.827,106.705,384.453,166.944,53.686,159.866
C07966=1017.834,106.987,384.433,166.947,53.677,159.865
C07967=1017.839,107.269,384.413,166.950,53.668,159.864
C07968=1017.845,107.551,384.392,166.954,53.658,159.863
C07969=1017.850,107.800,384.375,166.956,53.649,159.861
C07970=1017.855,108.050,384.357,166.959,53.641,159.860
C07971=1017.860,108.299,384.338,166.961,53.633,159.859
C07972=1017.865,108.549,384.322,166.965,53.624,159.858
C07973=1017.870,108.798,384.303,166.968,53.616,159.857
C07974=1017.875,109.047,384.286,166.970,53.607,159.856
C07975=1017.880,109.296,384.268,166.974,53.599,159.855
C07976=1017.886,109.545,384.250,166.976,53.591,159.854
C07977=1017.891,109.795,384.231,166.979,53.582,159.853
C07978=1017.896,110.044,384.213,166.982,53.574,159.852
C07979=1017.901,110.293,384.194,166.985,53.566,159.851
C07980=1017.906,110.543,384.177,166.988,53.558,159.850
C07981=1017.911,110.792,384.159,166.991,53.549,159.849
C07982=1017.916,111.041,384.141,166.993,53.541,159.848
C07983=1017.921,111.291,384.122,166.997,53.533,159.847
C07984=1017.926,111.540,384.105,166.999,53.524,159.845
C07985=1017.932,111.790,384.086,167.003,53.516,159.845
C07986=1017.937,112.038,384.067,167.005,53.508,159.843
C07987=1017.942,112.288,384.049,167.009,53.499,159.843
C07988=1017.946,112.537,384.031,167.011,53.491,159.841
C07989=1017.951,112.786,384.013,167.013,53.483,159.840
C07990=1017.956,113.035,383.994,167.017,53.475,159.839
C07991=1017.961,113.285,383.976,167.019,53.467,159.838
C07992=1017.966,113.535,383.957,167.023,53.458,159.837
C07993=1017.971,113.784,383.939,167.025,53.451,159.836
C07994=1017.976,114.033,383.920,167.029,53.442,159.835
C07995=1017.981,114.282,383.902,167.031,53.434,159.834
C07996=1017.986,114.531,383.884,167.033,53.426,159.833
C07997=1017.991,114.780,383.865,167.037,53.417,159.832
C07998=1017.996,115.030,383.847,167.039,53.410,159.831
C07999=1018.001,115.279,383.828,167.043,53.401,159.830
C08000=1018.006,115.528,383.810,167.045,53.393,159.829
C08001=1018.011,115.778,383.791,167.049,53.384,159.828
C08002=1018.016,116.026,383.773,167.051,53.377,159.827
C08003=1018.021,116.276,383.754,167.055,53.368,159.826
C08004=1018.026,116.526,383.736,167.057,53.360,159.825
C08005=1018.031,116.774,383.717,167.061,53.352,159.824
C08006=1018.035,117.024,383.698,167.063,53.343,159.823
C08007=1018.040,117.273,383.679,167.066,53.335,159.822
C08008=1018.045,117.522,383.661,167.069,53.327,159.821
C08009=1018.051,117.772,383.643,167.072,53.319,159.820
C08010=1018.056,118.021,383.624,167.074,53.310,159.819
C08011=1018.060,118.270,383.606,167.078,53.302,159.818
C08012=1018.066,118.519,383.587,167.081,53.294,159.817
C08013=1018.071,118.769,383.568,167.084,53.286,159.816
C08014=1018.076,119.018,383.549,167.087,53.278,159.815
C08015=1018.081,119.267,383.531,167.090,53.269,159.814
C08016=1018.086,119.517,383.513,167.092,53.261,159.813
C08017=1018.091,119.766,383.494,167.096,53.253,159.812
C08018=1018.096,120.015,383.476,167.099,53.245,159.811
C08019=1018.101,120.264,383.457,167.102,53.236,159.810
C08020=1018.106,120.513,383.439,167.104,53.228,159.809
C08021=1018.112,120.763,383.419,167.108,53.220,159.808
C08022=1018.116,121.012,383.401,167.110,53.212,159.807
C08023=1018.121,121.261,383.382,167.113,53.203,159.805
C08024=1018.126,121.510,383.364,167.116,53.195,159.804
C08025=1018.132,121.760,383.345,167.120,53.187,159.804
C08026=1018.137,122.009,383.327,167.122,53.179,159.802
C08027=1018.141,122.258,383.307,167.125,53.170,159.801
C08028=1018.146,122.508,383.289,167.128,53.163,159.800
C08029=1018.152,122.789,383.268,167.132,53.153,159.799
C08030=1018.158,123.071,383.247,167.135,53.144,159.798
C08031=1018.163,123.353,383.226,167.139,53.134,159.797
C08032=1018.169,123.635,383.205,167.142,53.125,159.796
C08033=1018.175,123.885,383.185,167.145,53.116,159.795
C08034=1018.180,124.134,383.167,167.148,53.109,159.794
C08035=1018.185,124.383,383.148,167.151,53.100,159.792
C08036=1018.191,124.632,383.129,167.153,53.092,159.791
C08037=1018.195,124.882,383.111,167.157,53.084,159.791
C08038=1018.201,125.130,383.092,167.160,53.075,159.789
C08039=1018.206,125.380,383.073,167.163,53.067,159.788
C08040=1018.211,125.629,383.055,167.166,53.059,159.787
C08041=1018.215,125.878,383.035,167.169,53.050,159.786
C08042=1018.221,126.128,383.017,167.172,53.042,159.785
C08043=1018.226,126.377,382.998,167.176,53.034,159.784
C08044=1018.231,126.626,382.979,167.178,53.025,159.783
C08045=1018.236,126.876,382.960,167.182,53.017,159.782
C08046=1018.241,127.125,382.941,167.184,53.009,159.781
C08047=1018.247,127.375,382.923,167.187,53.000,159.780
C08048=1018.252,127.623,382.904,167.191,52.992,159.779
C08049=1018.257,127.872,382.885,167.194,52.984,159.778
C08050=1018.263,128.122,382.866,167.197,52.975,159.777
C08051=1018.267,128.371,382.848,167.200,52.967,159.776
C08052=1018.273,128.620,382.828,167.203,52.959,159.775
C08053=1018.278,128.869,382.810,167.206,52.950,159.774
C08054=1018.283,129.118,382.791,167.209,52.942,159.773
C08055=1018.289,129.368,382.772,167.212,52.933,159.772
C08056=1018.293,129.617,382.753,167.216,52.925,159.771
C08057=1018.299,129.866,382.733,167.218,52.917,159.770
C08058=1018.303,130.116,382.715,167.222,52.909,159.769
C08059=1018.308,130.365,382.695,167.224,52.901,159.768
C08060=1018.314,130.614,382.677,167.228,52.892,159.767
C08061=1018.318,130.864,382.657,167.230,52.885,159.766
C08062=1018.324,131.113,382.638,167.234,52.876,159.765
C08063=1018.329,131.361,382.619,167.238,52.868,159.764
C08064=1018.334,131.611,382.599,167.240,52.860,159.763
C08065=1018.339,131.860,382.580,167.243,52.852,159.762
C08066=1018.344,132.110,382.560,167.246,52.844,159.761
C08067=1018.349,132.358,382.542,167.250,52.836,159.760
C08068=1018.354,132.608,382.522,167.252,52.828,159.759
C08069=1018.359,132.857,382.503,167.255,52.819,159.758
C08070=1018.364,133.107,382.484,167.259,52.811,159.757
C08071=1018.368,133.356,382.465,167.262,52.803,159.756
C08072=1018.374,133.605,382.446,167.265,52.795,159.755
C08073=1018.379,133.854,382.426,167.268,52.786,159.754
C08074=1018.384,134.104,382.407,167.271,52.778,159.753
C08075=1018.389,134.352,382.388,167.274,52.770,159.752
C08076=1018.394,134.602,382.368,167.278,52.762,159.751
C08077=1018.399,134.851,382.349,167.281,52.754,159.750
C08078=1018.404,135.101,382.329,167.283,52.745,159.749
C08079=1018.410,135.349,382.310,167.287,52.737,159.748
C08080=1018.415,135.599,382.290,167.290,52.729,159.747
C08081=1018.420,135.847,382.271,167.293,52.721,159.746
C08082=1018.425,136.097,382.251,167.297,52.712,159.745
C08083=1018.430,136.346,382.232,167.299,52.705,159.744
C08084=1018.435,136.596,382.213,167.303,52.696,159.743
C08085=1018.440,136.844,382.194,167.306,52.689,159.742
C08086=1018.445,137.094,382.174,167.309,52.680,159.741
C08087=1018.450,137.343,382.155,167.313,52.672,159.740
C08088=1018.455,137.592,382.135,167.315,52.664,159.739
C08089=1018.460,137.841,382.116,167.319,52.656,159.738
C08090=1018.465,138.090,382.096,167.322,52.648,159.737
C08091=1018.470,138.339,382.077,167.325,52.640,159.736
C08092=1018.475,138.589,382.057,167.329,52.631,159.735
C08093=1018.481,138.870,382.035,167.332,52.622,159.733
C08094=1018.486,139.152,382.012,167.335,52.613,159.732
C08095=1018.493,139.434,381.990,167.339,52.604,159.731
C08096=1018.498,139.717,381.968,167.343,52.595,159.730
C08097=1018.503,139.965,381.948,167.346,52.586,159.729
C08098=1018.508,140.215,381.928,167.350,52.578,159.728
C08099=1018.513,140.463,381.909,167.352,52.570,159.727
C08100=1018.518,140.713,381.889,167.356,52.562,159.726
C08101=1018.523,140.962,381.869,167.359,52.554,159.725
C08102=1018.527,141.211,381.849,167.362,52.546,159.724
C08103=1018.533,141.461,381.830,167.366,52.538,159.723
C08104=1018.538,141.709,381.810,167.368,52.530,159.722
C08105=1018.543,141.959,381.790,167.372,52.522,159.721
C08106=1018.548,142.208,381.771,167.375,52.514,159.720
C08107=1018.553,142.457,381.751,167.378,52.506,159.719
C08108=1018.558,142.707,381.731,167.382,52.498,159.718
C08109=1018.563,142.955,381.712,167.385,52.490,159.717
C08110=1018.568,143.204,381.691,167.388,52.481,159.716
C08111=1018.573,143.454,381.672,167.392,52.473,159.715
C08112=1018.579,143.702,381.652,167.394,52.465,159.714
C08113=1018.584,143.952,381.632,167.398,52.457,159.713
C08114=1018.588,144.202,381.612,167.402,52.449,159.713
C08115=1018.593,144.450,381.592,167.404,52.440,159.711
C08116=1018.599,144.700,381.573,167.408,52.432,159.710
C08117=1018.604,144.949,381.552,167.411,52.425,159.709
C08118=1018.608,145.198,381.533,167.414,52.416,159.708
C08119=1018.614,145.447,381.514,167.418,52.408,159.708
C08120=1018.619,145.696,381.493,167.420,52.400,159.706
C08121=1018.624,145.945,381.474,167.424,52.392,159.705
C08122=1018.629,146.194,381.453,167.428,52.384,159.705
C08123=1018.634,146.444,381.432,167.430,52.376,159.703
C08124=1018.639,146.693,381.413,167.434,52.368,159.703
C08125=1018.645,146.941,381.393,167.438,52.360,159.702
C08126=1018.650,147.191,381.373,167.441,52.352,159.701
C08127=1018.655,147.440,381.353,167.444,52.344,159.700
C08128=1018.659,147.689,381.333,167.448,52.336,159.699
C08129=1018.667,148.078,381.301,167.453,52.323,159.697
C08130=1018.675,148.468,381.269,167.457,52.310,159.696
C08131=1018.683,148.857,381.238,167.464,52.298,159.694
C08132=1018.691,149.246,381.207,167.468,52.285,159.693
C08133=1018.696,149.495,381.187,167.472,52.277,159.692
C08134=1018.701,149.744,381.167,167.475,52.270,159.691
C08135=1018.706,149.993,381.146,167.479,52.262,159.690
C08136=1018.711,150.242,381.126,167.482,52.253,159.689
C08137=1018.716,150.492,381.106,167.485,52.246,159.688
C08138=1018.721,150.740,381.085,167.489,52.238,159.687
C08139=1018.726,150.990,381.066,167.492,52.229,159.686
C08140=1018.731,151.239,381.045,167.495,52.221,159.685
C08141=1018.736,151.488,381.025,167.499,52.213,159.684
C08142=1018.741,151.737,381.004,167.502,52.205,159.683
C08143=1018.746,151.986,380.984,167.505,52.197,159.682
C08144=1018.751,152.235,380.964,167.509,52.189,159.681
C08145=1018.756,152.484,380.943,167.513,52.181,159.680
C08146=1018.762,152.733,380.923,167.515,52.173,159.679
C08147=1018.767,152.983,380.903,167.519,52.165,159.678
C08148=1018.771,153.232,380.883,167.523,52.157,159.677
C08149=1018.776,153.481,380.862,167.526,52.150,159.676
C08150=1018.782,153.730,380.842,167.529,52.141,159.675
C08151=1018.786,153.979,380.821,167.533,52.133,159.674
C08152=1018.791,154.228,380.800,167.536,52.125,159.673
C08153=1018.799,154.619,380.769,167.542,52.113,159.672
C08154=1018.807,155.010,380.736,167.547,52.100,159.670
C08155=1018.815,155.401,380.704,167.553,52.088,159.669
C08156=1018.823,155.792,380.672,167.557,52.075,159.668
C08157=1018.828,156.042,380.651,167.561,52.067,159.667
C08158=1018.833,156.290,380.631,167.565,52.059,159.666
C08159=1018.838,156.539,380.610,167.569,52.051,159.665
C08160=1018.843,156.788,380.590,167.572,52.044,159.664
C08161=1018.848,157.037,380.569,167.575,52.035,159.663
C08162=1018.853,157.287,380.548,167.579,52.027,159.662
C08163=1018.858,157.536,380.528,167.582,52.019,159.661
C08164=1018.863,157.785,380.507,167.585,52.011,159.660
C08165=1018.869,158.034,380.486,167.589,52.003,159.659
C08166=1018.874,158.283,380.466,167.593,51.995,159.658
C08167=1018.879,158.532,380.446,167.596,51.987,159.657
C08168=1018.883,158.781,380.425,167.600,51.979,159.656
C08169=1018.888,159.030,380.404,167.603,51.971,159.655
C08170=1018.893,159.279,380.382,167.607,51.964,159.654
C08171=1018.898,159.528,380.362,167.610,51.956,159.654
C08172=1018.903,159.778,380.340,167.614,51.948,159.653
C08173=1018.908,160.027,380.320,167.617,51.940,159.652
C08174=1018.913,160.276,380.298,167.621,51.932,159.651
C08175=1018.918,160.525,380.277,167.624,51.925,159.650
C08176=1018.922,160.773,380.257,167.628,51.917,159.649
C08177=1018.927,161.023,380.236,167.632,51.909,159.648
C08178=1018.932,161.271,380.214,167.634,51.902,159.647
C08179=1018.937,161.521,380.193,167.638,51.894,159.646
C08180=1018.941,161.770,380.172,167.642,51.886,159.645
C08181=1018.947,162.019,380.151,167.645,51.878,159.644
C08182=1018.951,162.268,380.130,167.649,51.871,159.644
C08183=1018.956,162.518,380.108,167.653,51.863,159.643
C08184=1018.962,162.766,380.087,167.656,51.855,159.642
C08185=1018.966,163.016,380.066,167.660,51.847,159.641
C08186=1018.972,163.264,380.045,167.663,51.839,159.640
C08187=1018.976,163.514,380.024,167.666,51.831,159.639
C08188=1018.981,163.763,380.002,167.670,51.824,159.638
C08189=1018.986,164.011,379.981,167.674,51.816,159.637
C08190=1018.991,164.261,379.960,167.677,51.808,159.636
C08191=1018.996,164.509,379.939,167.681,51.800,159.635
C08192=1019.001,164.759,379.918,167.685,51.792,159.634
C08193=1019.005,165.008,379.896,167.688,51.785,159.633
C08194=1019.011,165.257,379.875,167.691,51.777,159.632
C08195=1019.015,165.506,379.854,167.696,51.769,159.632
C08196=1019.021,165.755,379.833,167.700,51.761,159.631
C08197=1019.025,166.004,379.812,167.702,51.754,159.630
C08198=1019.030,166.253,379.790,167.706,51.746,159.629
C08199=1019.036,166.502,379.769,167.710,51.738,159.628
C08200=1019.040,166.751,379.747,167.714,51.730,159.627
C08201=1019.045,167.000,379.726,167.717,51.722,159.626
C08202=1019.050,167.249,379.705,167.721,51.715,159.625
C08203=1019.055,167.498,379.684,167.725,51.707,159.625
C08204=1019.061,167.747,379.663,167.729,51.699,159.624
C08205=1019.065,167.996,379.641,167.732,51.691,159.623
C08206=1019.070,168.245,379.620,167.735,51.683,159.622
C08207=1019.075,168.494,379.599,167.739,51.675,159.621
C08208=1019.080,168.743,379.577,167.743,51.667,159.620
C08209=1019.085,168.992,379.557,167.746,51.660,159.619
C08210=1019.091,169.242,379.534,167.750,51.652,159.618
C08211=1019.095,169.491,379.513,167.754,51.644,159.617
C08212=1019.101,169.740,379.492,167.758,51.636,159.616
C08213=1019.106,169.988,379.470,167.762,51.628,159.616
C08214=1019.110,170.238,379.449,167.765,51.621,159.615
C08215=1019.116,170.486,379.428,167.769,51.613,159.614
C08216=1019.120,170.736,379.406,167.772,51.605,159.613
C08217=1019.126,171.017,379.382,167.777,51.596,159.612
C08218=1019.132,171.299,379.358,167.781,51.587,159.611
C08219=1019.138,171.580,379.333,167.785,51.579,159.610
C08220=1019.143,171.862,379.309,167.790,51.570,159.609
C08221=1019.148,172.111,379.288,167.794,51.562,159.608
C08222=1019.154,172.359,379.266,167.798,51.554,159.607
C08223=1019.158,172.609,379.245,167.801,51.546,159.606
C08224=1019.164,172.858,379.223,167.804,51.538,159.605
C08225=1019.169,173.107,379.202,167.808,51.531,159.604
C08226=1019.174,173.356,379.181,167.812,51.523,159.603
C08227=1019.179,173.605,379.159,167.816,51.515,159.602
C08228=1019.184,173.853,379.137,167.820,51.507,159.602
C08229=1019.190,174.103,379.115,167.824,51.499,159.601
C08230=1019.195,174.352,379.095,167.828,51.491,159.600
C08231=1019.200,174.601,379.073,167.831,51.484,159.599
C08232=1019.205,174.850,379.051,167.835,51.476,159.598
C08233=1019.211,175.099,379.029,167.839,51.468,159.597
C08234=1019.215,175.348,379.008,167.843,51.460,159.596
C08235=1019.220,175.597,378.986,167.846,51.452,159.595
C08236=1019.226,175.846,378.965,167.850,51.444,159.594
C08237=1019.231,176.095,378.943,167.855,51.437,159.594
C08238=1019.236,176.344,378.921,167.859,51.429,159.593
C08239=1019.241,176.593,378.900,167.862,51.421,159.592
C08240=1019.246,176.842,378.878,167.866,51.413,159.591
C08241=1019.251,177.091,378.856,167.870,51.405,159.590
C08242=1019.257,177.340,378.835,167.874,51.397,159.589
C08243=1019.262,177.589,378.813,167.877,51.390,159.588
C08244=1019.268,177.838,378.791,167.881,51.382,159.587
C08245=1019.273,178.087,378.770,167.885,51.374,159.586
C08246=1019.277,178.336,378.748,167.889,51.367,159.586
C08247=1019.283,178.585,378.727,167.893,51.359,159.585
C08248=1019.288,178.834,378.705,167.897,51.351,159.584
C08249=1019.293,179.083,378.683,167.901,51.343,159.583
C08250=1019.299,179.331,378.662,167.905,51.335,159.582
C08251=1019.304,179.581,378.640,167.909,51.327,159.581
C08252=1019.309,179.830,378.618,167.913,51.319,159.580
C08253=1019.315,180.079,378.596,167.917,51.311,159.579
C08254=1019.320,180.328,378.574,167.921,51.303,159.578
C08255=1019.325,180.577,378.552,167.924,51.295,159.577
C08256=1019.331,180.826,378.531,167.929,51.288,159.577
C08257=1019.336,181.075,378.509,167.933,51.280,159.576
C08258=1019.341,181.323,378.487,167.937,51.272,159.575
C08259=1019.347,181.573,378.465,167.941,51.264,159.574
C08260=1019.352,181.821,378.444,167.945,51.256,159.573
C08261=1019.357,182.071,378.421,167.948,51.249,159.572
C08262=1019.362,182.320,378.399,167.953,51.241,159.572
C08263=1019.367,182.569,378.377,167.957,51.233,159.571
C08264=1019.372,182.818,378.354,167.961,51.226,159.570
C08265=1019.376,183.067,378.332,167.965,51.218,159.569
C08266=1019.382,183.316,378.310,167.969,51.210,159.568
C08267=1019.386,183.565,378.287,167.972,51.204,159.567
C08268=1019.392,183.814,378.265,167.976,51.196,159.566
C08269=1019.396,184.063,378.243,167.981,51.189,159.566
C08270=1019.401,184.312,378.219,167.984,51.181,159.565
C08271=1019.406,184.561,378.197,167.989,51.173,159.564
C08272=1019.411,184.809,378.175,167.993,51.166,159.563
C08273=1019.416,185.058,378.153,167.997,51.158,159.562
C08274=1019.421,185.308,378.130,168.001,51.150,159.562
C08275=1019.426,185.556,378.107,168.004,51.143,159.561
C08276=1019.431,185.806,378.085,168.008,51.136,159.560
C08277=1019.436,186.054,378.062,168.012,51.128,159.559
C08278=1019.441,186.304,378.040,168.017,51.121,159.558
C08279=1019.446,186.552,378.017,168.021,51.113,159.557
C08280=1019.451,186.802,377.994,168.025,51.105,159.556
C08281=1019.457,187.082,377.969,168.030,51.097,159.556
C08282=1019.462,187.363,377.944,168.034,51.088,159.555
C08283=1019.468,187.644,377.918,168.039,51.080,159.554
C08284=1019.474,187.925,377.893,168.043,51.071,159.553
C08285=1019.479,188.174,377.870,168.047,51.064,159.552
C08286=1019.484,188.423,377.847,168.051,51.056,159.551
C08287=1019.489,188.672,377.825,168.055,51.049,159.550
C08288=1019.494,188.921,377.802,168.059,51.041,159.550
C08289=1019.499,189.170,377.780,168.063,51.033,159.549
C08290=1019.505,189.419,377.757,168.068,51.026,159.548
C08291=1019.509,189.668,377.735,168.072,51.018,159.547
C08292=1019.514,189.917,377.712,168.076,51.011,159.546
C08293=1019.520,190.165,377.689,168.080,51.003,159.545
C08294=1019.525,190.415,377.667,168.084,50.996,159.545
C08295=1019.530,190.664,377.643,168.088,50.988,159.544
C08296=1019.535,190.912,377.621,168.093,50.981,159.543
C08297=1019.541,191.162,377.598,168.097,50.973,159.542
C08298=1019.545,191.410,377.575,168.101,50.965,159.541
C08299=1019.550,191.660,377.553,168.105,50.958,159.541
C08300=1019.556,191.908,377.530,168.109,50.950,159.540
C08301=1019.561,192.157,377.507,168.113,50.943,159.539
C08302=1019.566,192.406,377.484,168.118,50.935,159.538
C08303=1019.571,192.655,377.462,168.123,50.928,159.537
C08304=1019.576,192.904,377.439,168.127,50.920,159.537
C08305=1019.581,193.152,377.416,168.131,50.913,159.536
C08306=1019.587,193.402,377.394,168.135,50.905,159.535
C08307=1019.592,193.651,377.370,168.140,50.898,159.534
C08308=1019.597,193.899,377.348,168.144,50.890,159.533
C08309=1019.602,194.148,377.325,168.148,50.882,159.532
C08310=1019.607,194.398,377.302,168.152,50.875,159.532
C08311=1019.612,194.646,377.279,168.156,50.867,159.531
C08312=1019.618,194.895,377.256,168.160,50.860,159.530
C08313=1019.623,195.144,377.233,168.164,50.852,159.529
C08314=1019.628,195.392,377.210,168.169,50.845,159.528
C08315=1019.634,195.642,377.188,168.174,50.837,159.528
C08316=1019.639,195.891,377.164,168.178,50.830,159.527
C08317=1019.644,196.140,377.141,168.182,50.822,159.526
C08318=1019.649,196.388,377.119,168.186,50.815,159.525
C08319=1019.654,196.637,377.095,168.190,50.807,159.524
C08320=1019.660,196.886,377.072,168.195,50.800,159.524
C08321=1019.665,197.134,377.050,168.199,50.792,159.523
C08322=1019.670,197.384,377.026,168.204,50.784,159.522
C08323=1019.676,197.633,377.004,168.208,50.777,159.521
C08324=1019.681,197.882,376.981,168.212,50.769,159.520
C08325=1019.686,198.131,376.958,168.217,50.762,159.520
C08326=1019.692,198.379,376.935,168.221,50.754,159.519
C08327=1019.697,198.628,376.912,168.225,50.747,159.518
C08328=1019.702,198.878,376.888,168.230,50.739,159.517
C08329=1019.708,199.126,376.866,168.235,50.731,159.517
C08330=1019.713,199.375,376.843,168.239,50.724,159.516
C08331=1019.718,199.624,376.819,168.243,50.717,159.515
C08332=1019.723,199.873,376.796,168.247,50.709,159.514
C08333=1019.729,200.122,376.773,168.251,50.702,159.513
C08334=1019.734,200.371,376.749,168.256,50.695,159.513
C08335=1019.739,200.619,376.726,168.260,50.687,159.512
C08336=1019.744,200.868,376.703,168.265,50.679,159.511
C08337=1019.749,201.117,376.679,168.270,50.672,159.510
C08338=1019.755,201.366,376.655,168.274,50.665,159.510
C08339=1019.760,201.615,376.631,168.278,50.657,159.509
C08340=1019.765,201.863,376.609,168.283,50.650,159.508
C08341=1019.770,202.112,376.585,168.287,50.643,159.507
C08342=1019.775,202.361,376.561,168.291,50.635,159.506
C08343=1019.781,202.610,376.538,168.297,50.628,159.506
C08344=1019.786,202.859,376.514,168.301,50.621,159.505
C08345=1019.807,203.899,376.416,168.755,50.715,159.604
C08346=1019.812,204.119,376.394,168.758,50.709,159.603
C08347=1019.818,204.340,376.371,168.762,50.703,159.602
C08348=1019.824,204.561,376.349,168.765,50.698,159.602
C08349=1019.829,204.781,376.327,168.768,50.692,159.601
C08350=1019.835,205.003,376.305,168.771,50.686,159.600
C08351=1019.841,205.224,376.282,168.775,50.680,159.600
C08352=1019.846,205.444,376.260,168.778,50.675,159.599
C08353=1019.851,205.665,376.238,168.781,50.669,159.598
C08354=1019.857,205.914,376.213,168.784,50.663,159.598
C08355=1019.864,206.163,376.187,168.789,50.656,159.597
C08356=1019.869,206.412,376.161,168.793,50.650,159.596
C08357=1019.875,206.660,376.136,168.796,50.644,159.595
C08358=1019.881,206.908,376.111,168.800,50.637,159.595
C08359=1019.887,207.157,376.086,168.803,50.631,159.594
C08360=1019.893,207.406,376.060,168.807,50.625,159.593
C08361=1019.900,207.654,376.035,168.810,50.619,159.593
C08362=1019.906,207.903,376.010,168.814,50.613,159.592
C08363=1019.912,208.152,375.984,168.818,50.606,159.591
C08364=1019.918,208.400,375.959,168.821,50.600,159.590
C08365=1019.924,208.649,375.934,168.825,50.594,159.590
C08366=1019.931,208.898,375.908,168.829,50.588,159.589
C08367=1019.937,209.146,375.883,168.833,50.582,159.589
C08368=1019.943,209.395,375.858,168.836,50.575,159.588
C08369=1019.948,209.644,375.832,168.840,50.569,159.587
C08370=1019.955,209.893,375.806,168.843,50.563,159.586
C08371=1019.961,210.141,375.781,168.847,50.557,159.586
C08372=1019.966,210.389,375.756,168.851,50.551,159.585
C08373=1019.973,210.638,375.731,168.855,50.545,159.584
C08374=1019.978,210.886,375.704,168.858,50.538,159.584
C08375=1019.985,211.135,375.679,168.862,50.532,159.583
C08376=1019.991,211.384,375.653,168.866,50.526,159.582
C08377=1019.996,211.633,375.628,168.869,50.520,159.582
C08378=1020.003,211.881,375.602,168.873,50.514,159.581
C08379=1020.009,212.129,375.576,168.877,50.508,159.580
C08380=1020.015,212.378,375.550,168.881,50.502,159.580
C08381=1020.021,212.627,375.525,168.884,50.496,159.579
C08382=1020.027,212.876,375.500,168.888,50.490,159.578
C08383=1020.033,213.124,375.473,168.892,50.484,159.578
C08384=1020.039,213.373,375.448,168.895,50.478,159.577
C08385=1020.045,213.621,375.422,168.898,50.472,159.576
C08386=1020.052,213.869,375.396,168.902,50.466,159.576
C08387=1020.057,214.118,375.370,168.906,50.460,159.575
C08388=1020.064,214.368,375.344,168.910,50.454,159.574
C08389=1020.070,214.616,375.318,168.914,50.448,159.574
C08390=1020.076,214.865,375.293,168.917,50.442,159.573
C08391=1020.082,215.113,375.267,168.921,50.436,159.572
C08392=1020.089,215.361,375.241,168.925,50.430,159.572
C08393=1020.095,215.610,375.216,168.929,50.424,159.571
C08394=1020.100,215.859,375.190,168.932,50.417,159.570
C08395=1020.107,216.107,375.164,168.937,50.412,159.570
C08396=1020.113,216.356,375.138,168.940,50.406,159.569
C08397=1020.118,216.605,375.113,168.944,50.400,159.569
C08398=1020.125,216.853,375.086,168.948,50.394,159.568
C08399=1020.132,217.102,375.061,168.952,50.388,159.567
C08400=1020.138,217.351,375.034,168.955,50.382,159.567
C08401=1020.144,217.599,375.009,168.959,50.376,159.566
C08402=1020.150,217.847,374.983,168.962,50.370,159.565
C08403=1020.156,218.096,374.957,168.966,50.365,159.565
C08404=1020.162,218.344,374.931,168.970,50.359,159.564
C08405=1020.168,218.593,374.905,168.974,50.353,159.563
C08406=1020.177,218.962,374.867,168.980,50.345,159.563
C08407=1020.186,219.331,374.828,168.985,50.336,159.562
C08408=1020.195,219.700,374.789,168.990,50.328,159.561
C08409=1020.205,220.068,374.749,168.996,50.319,159.560
C08410=1020.210,220.317,374.723,169.000,50.313,159.559
C08411=1020.216,220.566,374.697,169.004,50.307,159.559
C08412=1020.222,220.814,374.671,169.008,50.302,159.558
C08413=1020.228,221.063,374.645,169.011,50.296,159.557
C08414=1020.235,221.312,374.618,169.015,50.291,159.557
C08415=1020.241,221.560,374.592,169.019,50.285,159.556
C08416=1020.246,221.809,374.566,169.023,50.279,159.556
C08417=1020.253,222.057,374.540,169.027,50.273,159.555
C08418=1020.258,222.305,374.513,169.031,50.267,159.555
C08419=1020.265,222.555,374.487,169.035,50.262,159.554
C08420=1020.271,222.803,374.461,169.038,50.256,159.553
C08421=1020.277,223.051,374.434,169.042,50.251,159.553
C08422=1020.283,223.299,374.408,169.046,50.245,159.552
C08423=1020.290,223.548,374.381,169.050,50.240,159.552
C08424=1020.296,223.797,374.356,169.054,50.234,159.551
C08425=1020.302,224.045,374.329,169.058,50.228,159.551
C08426=1020.307,224.294,374.302,169.061,50.223,159.550
C08427=1020.315,224.543,374.276,169.065,50.217,159.550
C08428=1020.320,224.791,374.249,169.069,50.211,159.549
C08429=1020.326,225.040,374.223,169.073,50.206,159.548
C08430=1020.332,225.288,374.197,169.077,50.200,159.548
C08431=1020.339,225.537,374.170,169.081,50.195,159.547
C08432=1020.345,225.785,374.144,169.084,50.189,159.547
C08433=1020.351,226.033,374.118,169.088,50.184,159.546
C08434=1020.357,226.283,374.091,169.091,50.178,159.545
C08435=1020.364,226.531,374.064,169.096,50.173,159.545
C08436=1020.370,226.779,374.038,169.100,50.167,159.544
C08437=1020.375,227.027,374.011,169.104,50.161,159.544
C08438=1020.382,227.276,373.984,169.107,50.156,159.543
C08439=1020.388,227.524,373.958,169.111,50.151,159.543
C08440=1020.394,227.773,373.931,169.115,50.146,159.542
C08441=1020.400,228.022,373.904,169.119,50.140,159.542
C08442=1020.406,228.270,373.878,169.123,50.134,159.541
C08443=1020.412,228.519,373.851,169.126,50.129,159.541
C08444=1020.418,228.768,373.824,169.131,50.124,159.540
C08445=1020.424,229.016,373.797,169.134,50.118,159.540
C08446=1020.432,229.342,373.762,169.139,50.112,159.539
C08447=1020.441,229.670,373.727,169.145,50.104,159.538
C08448=1020.449,229.996,373.692,169.150,50.097,159.538
C08449=1020.457,230.322,373.657,169.155,50.090,159.537
C08450=1020.463,230.571,373.630,169.159,50.085,159.536
C08451=1020.469,230.820,373.603,169.163,50.080,159.536
C08452=1020.475,231.067,373.576,169.166,50.075,159.535
C08453=1020.481,231.317,373.549,169.170,50.069,159.535
C08454=1020.487,231.565,373.522,169.174,50.064,159.534
C08455=1020.493,231.813,373.495,169.179,50.059,159.534
C08456=1020.500,232.062,373.468,169.182,50.054,159.533
C08457=1020.505,232.310,373.441,169.186,50.048,159.533
C08458=1020.512,232.559,373.414,169.190,50.043,159.533
C08459=1020.518,232.807,373.387,169.194,50.038,159.532
C08460=1020.524,233.056,373.360,169.198,50.033,159.532
C08461=1020.530,233.304,373.333,169.202,50.028,159.531
C08462=1020.535,233.524,373.309,169.205,50.023,159.531
C08463=1020.540,233.743,373.285,169.209,50.018,159.530
C08464=1020.546,233.963,373.261,169.212,50.014,159.530
C08465=1020.551,234.183,373.237,169.215,50.009,159.529
C08466=1020.557,234.402,373.213,169.219,50.005,159.529
C08467=1020.562,234.621,373.189,169.223,49.999,159.528
C08468=1020.568,234.841,373.165,169.227,49.995,159.528
C08469=1020.573,235.060,373.141,169.230,49.991,159.528
C08470=1020.579,235.309,373.114,169.233,49.986,159.527
C08471=1020.586,235.557,373.086,169.238,49.981,159.527
C08472=1020.591,235.805,373.060,169.242,49.975,159.526
C08473=1020.598,236.054,373.033,169.246,49.970,159.526
C08474=1020.604,236.302,373.005,169.249,49.965,159.525
C08475=1020.610,236.551,372.978,169.253,49.960,159.525
C08476=1020.617,236.800,372.951,169.258,49.954,159.524
C08477=1020.623,237.048,372.924,169.261,49.950,159.524
C08478=1020.629,237.296,372.896,169.265,49.945,159.524
C08479=1020.635,237.545,372.870,169.270,49.940,159.523
C08480=1020.641,237.794,372.841,169.274,49.934,159.523
C08481=1020.647,238.042,372.815,169.277,49.929,159.522
C08482=1020.653,238.290,372.787,169.281,49.925,159.522
C08483=1020.660,238.538,372.760,169.286,49.919,159.521
C08484=1020.666,238.787,372.732,169.290,49.914,159.521
C08485=1020.673,239.036,372.705,169.293,49.909,159.520
C08486=1020.678,239.284,372.678,169.298,49.905,159.520
C08487=1020.685,239.532,372.650,169.302,49.899,159.520
C08488=1020.690,239.780,372.622,169.305,49.894,159.519
C08489=1020.697,240.029,372.595,169.310,49.890,159.519
C08490=1020.702,240.278,372.567,169.314,49.885,159.518
C08491=1020.709,240.526,372.540,169.317,49.880,159.518
C08492=1020.715,240.774,372.512,169.322,49.875,159.517
C08493=1020.721,241.022,372.484,169.326,49.870,159.517
C08494=1020.727,241.272,372.457,169.329,49.865,159.517
C08495=1020.733,241.519,372.430,169.334,49.860,159.516
C08496=1020.739,241.768,372.401,169.338,49.856,159.516
C08497=1020.746,242.016,372.374,169.341,49.851,159.515
C08498=1020.751,242.265,372.346,169.346,49.846,159.515
C08499=1020.758,242.513,372.318,169.350,49.841,159.515
C08500=1020.764,242.762,372.291,169.354,49.836,159.514
C08501=1020.770,243.010,372.263,169.358,49.831,159.514
C08502=1020.776,243.259,372.235,169.363,49.827,159.514
C08503=1020.782,243.506,372.208,169.366,49.822,159.513
C08504=1020.788,243.755,372.180,169.370,49.817,159.513
C08505=1020.794,244.004,372.151,169.374,49.812,159.512
C08506=1020.800,244.251,372.124,169.378,49.808,159.512
C08507=1020.806,244.500,372.096,169.383,49.803,159.512
C08508=1020.812,244.749,372.067,169.386,49.798,159.511
C08509=1020.818,244.997,372.040,169.391,49.793,159.511
C08510=1020.825,245.245,372.011,169.394,49.789,159.510
C08511=1020.830,245.494,371.982,169.398,49.784,159.510
C08512=1020.837,245.741,371.955,169.403,49.779,159.510
C08513=1020.843,245.990,371.927,169.407,49.775,159.509
C08514=1020.848,246.239,371.898,169.411,49.770,159.509
C08515=1020.855,246.487,371.871,169.414,49.766,159.508
C08516=1020.860,246.735,371.843,169.419,49.761,159.508
C08517=1020.866,246.984,371.814,169.423,49.756,159.508
C08518=1020.873,247.232,371.786,169.427,49.752,159.508
C08519=1020.879,247.480,371.758,169.431,49.747,159.507
C08520=1020.885,247.729,371.730,169.435,49.743,159.507
C08521=1020.891,247.977,371.702,169.439,49.738,159.507
C08522=1020.897,248.193,371.677,169.443,49.734,159.506
C08523=1020.902,248.410,371.653,169.447,49.730,159.506
C08524=1020.907,248.625,371.628,169.451,49.726,159.506
C08525=1020.912,248.842,371.604,169.454,49.722,159.505
C08526=1020.918,249.059,371.579,169.457,49.718,159.505
C08527=1020.923,249.275,371.554,169.461,49.714,159.505
C08528=1020.929,249.491,371.529,169.465,49.710,159.505
C08529=1020.934,249.707,371.505,169.468,49.706,159.504
C08530=1020.940,249.956,371.476,169.473,49.702,159.504
C08531=1020.947,250.204,371.449,169.476,49.697,159.504
C08532=1020.953,250.453,371.420,169.481,49.693,159.503
C08533=1020.958,250.701,371.392,169.485,49.688,159.503
C08534=1020.965,250.949,371.364,169.489,49.683,159.502
C08535=1020.971,251.197,371.335,169.493,49.679,159.502
C08536=1020.977,251.446,371.307,169.497,49.674,159.502
C08537=1020.984,251.694,371.279,169.502,49.670,159.501
C08538=1020.990,251.943,371.250,169.506,49.665,159.501
C08539=1020.996,252.191,371.221,169.510,49.661,159.501
C08540=1021.002,252.439,371.194,169.514,49.656,159.501
C08541=1021.008,252.687,371.166,169.518,49.652,159.500
C08542=1021.014,252.935,371.137,169.523,49.648,159.500
C08543=1021.021,253.184,371.109,169.527,49.643,159.500
C08544=1021.027,253.432,371.080,169.531,49.639,159.499
C08545=1021.033,253.681,371.052,169.535,49.634,159.499
C08546=1021.040,253.929,371.023,169.540,49.630,159.499
C08547=1021.046,254.177,370.995,169.543,49.625,159.498
C08548=1021.052,254.425,370.966,169.548,49.621,159.498
C08549=1021.059,254.674,370.938,169.552,49.617,159.498
C08550=1021.065,254.922,370.909,169.556,49.612,159.497
C08551=1021.071,255.171,370.881,169.561,49.607,159.497
C08552=1021.078,255.419,370.852,169.564,49.603,159.497
C08553=1021.084,255.667,370.824,169.569,49.599,159.497
C08554=1021.090,255.916,370.795,169.574,49.594,159.496
C08555=1021.096,256.164,370.766,169.577,49.590,159.496
C08556=1021.103,256.412,370.738,169.582,49.586,159.496
C08557=1021.110,256.660,370.709,169.586,49.582,159.495
C08558=1021.115,256.909,370.681,169.590,49.577,159.495
C08559=1021.122,257.157,370.652,169.595,49.573,159.495
C08560=1021.128,257.406,370.624,169.599,49.568,159.495
C08561=1021.135,257.654,370.595,169.603,49.564,159.494
C08562=1021.142,257.902,370.566,169.608,49.559,159.494
C08563=1021.148,258.150,370.538,169.612,49.556,159.494
C08564=1021.154,258.398,370.509,169.616,49.551,159.494
C08565=1021.161,258.646,370.481,169.621,49.547,159.493
C08566=1021.167,258.895,370.452,169.625,49.542,159.493
C08567=1021.173,259.143,370.423,169.629,49.538,159.493
C08568=1021.180,259.391,370.395,169.633,49.534,159.492
C08569=1021.186,259.639,370.366,169.638,49.530,159.492
C08570=1021.192,259.888,370.337,169.642,49.525,159.492
C08571=1021.198,260.136,370.308,169.646,49.521,159.492
C08572=1021.205,260.384,370.280,169.651,49.517,159.491
C08573=1021.211,260.632,370.250,169.654,49.513,159.491
C08574=1021.217,260.880,370.221,169.659,49.509,159.491
C08575=1021.223,261.128,370.192,169.664,49.504,159.491
C08576=1021.230,261.377,370.163,169.668,49.501,159.491
C08577=1021.237,261.625,370.134,169.673,49.496,159.490
C08578=1021.243,261.874,370.105,169.677,49.493,159.490
C08579=1021.249,262.122,370.076,169.681,49.488,159.490
C08580=1021.255,262.370,370.047,169.685,49.484,159.490
C08581=1021.262,262.618,370.018,169.690,49.480,159.489
C08582=1021.267,262.833,369.992,169.694,49.476,159.489
C08583=1021.272,263.049,369.967,169.698,49.473,159.489
C08584=1021.278,263.265,369.941,169.701,49.470,159.489
C08585=1021.283,263.480,369.915,169.705,49.466,159.489
C08586=1021.289,263.696,369.890,169.709,49.462,159.488
C08587=1021.294,263.911,369.865,169.713,49.459,159.488
C08588=1021.300,264.126,369.839,169.716,49.455,159.488
C08589=1021.305,264.342,369.814,169.720,49.452,159.488
C08590=1021.312,264.590,369.785,169.724,49.448,159.488
C08591=1021.318,264.838,369.756,169.729,49.444,159.488
C08592=1021.324,265.086,369.726,169.733,49.440,159.487
C08593=1021.330,265.334,369.697,169.738,49.436,159.487
C08594=1021.337,265.583,369.667,169.742,49.432,159.487
C08595=1021.343,265.831,369.638,169.747,49.428,159.487
C08596=1021.350,266.079,369.609,169.752,49.424,159.487
C08597=1021.356,266.327,369.580,169.755,49.420,159.486
C08598=1021.361,266.575,369.550,169.760,49.416,159.486
C08599=1021.368,266.824,369.521,169.764,49.412,159.486
C08600=1021.375,267.072,369.491,169.769,49.408,159.486
C08601=1021.381,267.320,369.462,169.773,49.404,159.486
C08602=1021.387,267.568,369.431,169.778,49.400,159.486
C08603=1021.394,267.817,369.402,169.782,49.397,159.485
C08604=1021.400,268.065,369.373,169.787,49.393,159.485
C08605=1021.406,268.313,369.343,169.791,49.389,159.485
C08606=1021.412,268.561,369.314,169.795,49.385,159.485
C08607=1021.419,268.809,369.283,169.800,49.381,159.485
C08608=1021.425,269.057,369.254,169.804,49.378,159.485
C08609=1021.431,269.305,369.225,169.809,49.374,159.484
C08610=1021.437,269.553,369.195,169.813,49.370,159.484
C08611=1021.444,269.802,369.166,169.818,49.366,159.484
C08612=1021.450,270.050,369.135,169.822,49.362,159.484
C08613=1021.457,270.297,369.105,169.827,49.358,159.484
C08614=1021.463,270.546,369.075,169.832,49.354,159.484
C08615=1021.469,270.794,369.046,169.835,49.351,159.483
C08616=1021.475,271.042,369.016,169.840,49.347,159.483
C08617=1021.482,271.290,368.986,169.844,49.343,159.483
C08618=1021.488,271.538,368.956,169.849,49.339,159.483
C08619=1021.494,271.786,368.927,169.853,49.336,159.483
C08620=1021.501,272.035,368.896,169.858,49.332,159.483
C08621=1021.507,272.283,368.867,169.862,49.328,159.483
C08622=1021.513,272.531,368.837,169.867,49.325,159.483
C08623=1021.520,272.779,368.806,169.871,49.321,159.482
C08624=1021.526,273.027,368.777,169.876,49.317,159.482
C08625=1021.532,273.276,368.747,169.881,49.314,159.482
C08626=1021.539,273.523,368.717,169.886,49.310,159.482
C08627=1021.545,273.771,368.686,169.891,49.307,159.482
C08628=1021.552,274.019,368.656,169.895,49.303,159.482
C08629=1021.557,274.268,368.627,169.899,49.299,159.482
C08630=1021.565,274.516,368.597,169.903,49.296,159.482
C08631=1021.570,274.764,368.566,169.908,49.292,159.482
C08632=1021.577,275.012,368.536,169.913,49.289,159.482
C08633=1021.583,275.260,368.506,169.918,49.285,159.482
C08634=1021.589,275.508,368.475,169.922,49.281,159.481
C08635=1021.596,275.756,368.445,169.927,49.278,159.481
C08636=1021.602,276.004,368.416,169.931,49.274,159.481
C08637=1021.609,276.252,368.386,169.936,49.271,159.481
C08638=1021.615,276.500,368.355,169.941,49.267,159.481
C08639=1021.622,276.748,368.325,169.945,49.263,159.481
C08640=1021.628,276.996,368.295,169.950,49.260,159.481
C08641=1021.634,277.245,368.264,169.954,49.257,159.481
C08642=1021.640,277.462,368.237,169.958,49.253,159.481
C08643=1021.645,277.680,368.210,169.963,49.250,159.481
C08644=1021.651,277.897,368.184,169.967,49.247,159.481
C08645=1021.656,278.115,368.157,169.971,49.244,159.481
C08646=1021.661,278.333,368.130,169.974,49.241,159.480
C08647=1021.668,278.550,368.103,169.978,49.238,159.480
C08648=1021.673,278.769,368.076,169.983,49.235,159.480
C08649=1021.679,278.987,368.050,169.987,49.232,159.480
C08650=1021.685,279.234,368.020,169.992,49.229,159.480
C08651=1021.691,279.483,367.989,169.996,49.225,159.480
C08652=1021.697,279.730,367.958,170.001,49.222,159.480
C08653=1021.704,279.979,367.927,170.005,49.218,159.480
C08654=1021.711,280.227,367.897,170.011,49.215,159.480
C08655=1021.717,280.475,367.867,170.015,49.212,159.480
C08656=1021.723,280.723,367.836,170.020,49.209,159.480
C08657=1021.729,280.970,367.805,170.024,49.205,159.480
C08658=1021.736,281.219,367.774,170.029,49.202,159.480
C08659=1021.743,281.467,367.744,170.033,49.198,159.480
C08660=1021.749,281.714,367.713,170.039,49.195,159.480
C08661=1021.756,281.963,367.682,170.043,49.192,159.480
C08662=1021.761,282.211,367.652,170.048,49.188,159.480
C08663=1021.768,282.459,367.621,170.053,49.184,159.480
C08664=1021.775,282.707,367.590,170.057,49.182,159.480
C08665=1021.781,282.955,367.560,170.063,49.178,159.480
C08666=1021.788,283.202,367.529,170.067,49.175,159.480
C08667=1021.794,283.451,367.498,170.072,49.172,159.480
C08668=1021.801,283.700,367.467,170.076,49.169,159.480
C08669=1021.807,283.946,367.437,170.081,49.165,159.480
C08670=1021.814,284.195,367.406,170.086,49.162,159.480
C08671=1021.821,284.443,367.375,170.091,49.159,159.480
C08672=1021.826,284.691,367.344,170.096,49.155,159.480
C08673=1021.833,284.939,367.313,170.100,49.152,159.480
C08674=1021.840,285.187,367.283,170.106,49.149,159.480
C08675=1021.846,285.435,367.251,170.110,49.145,159.480
C08676=1021.852,285.683,367.220,170.115,49.142,159.480
C08677=1021.859,285.931,367.189,170.119,49.139,159.480
C08678=1021.866,286.179,367.157,170.125,49.136,159.480
C08679=1021.872,286.427,367.127,170.129,49.133,159.480
C08680=1021.878,286.674,367.096,170.134,49.129,159.480
C08681=1021.885,286.922,367.064,170.139,49.126,159.480
C08682=1021.891,287.171,367.034,170.144,49.123,159.480
C08683=1021.898,287.419,367.002,170.149,49.120,159.480
C08684=1021.904,287.666,366.971,170.153,49.117,159.480
C08685=1021.911,287.914,366.940,170.159,49.114,159.480
C08686=1021.917,288.162,366.909,170.163,49.111,159.480
C08687=1021.924,288.410,366.877,170.168,49.108,159.480
C08688=1021.931,288.658,366.846,170.173,49.105,159.480
C08689=1021.937,288.905,366.815,170.178,49.102,159.480
C08690=1021.944,289.153,366.783,170.183,49.099,159.480
C08691=1021.950,289.402,366.753,170.188,49.096,159.480
C08692=1021.956,289.650,366.721,170.193,49.093,159.480
C08693=1021.963,289.898,366.689,170.197,49.090,159.481
C08694=1021.969,290.146,366.658,170.203,49.087,159.481
C08695=1021.976,290.394,366.626,170.207,49.084,159.481
C08696=1021.982,290.641,366.595,170.212,49.081,159.481
C08697=1021.989,290.889,366.564,170.218,49.077,159.481
C08698=1021.996,291.137,366.533,170.222,49.075,159.481
C08699=1022.002,291.385,366.501,170.227,49.071,159.481
C08700=1022.008,291.633,366.469,170.232,49.069,159.481
C08701=1022.015,291.881,366.438,170.237,49.065,159.481
C08702=1022.021,292.104,366.409,170.242,49.063,159.481
C08703=1022.027,292.329,366.381,170.246,49.060,159.481
C08704=1022.033,292.552,366.352,170.250,49.057,159.481
C08705=1022.039,292.776,366.324,170.255,49.055,159.481
C08706=1022.045,293.000,366.295,170.259,49.052,159.481
C08707=1022.050,293.224,366.267,170.264,49.049,159.481
C08708=1022.056,293.448,366.238,170.268,49.047,159.482
C08709=1022.062,293.672,366.209,170.273,49.044,159.482
C08710=1022.069,293.920,366.177,170.278,49.042,159.482
C08711=1022.075,294.168,366.145,170.283,49.039,159.482
C08712=1022.082,294.415,366.113,170.288,49.036,159.482
C08713=1022.088,294.664,366.081,170.293,49.034,159.482
C08714=1022.095,294.911,366.049,170.298,49.030,159.482
C08715=1022.101,295.159,366.017,170.303,49.028,159.482
C08716=1022.107,295.407,365.984,170.308,49.025,159.483
C08717=1022.114,295.655,365.953,170.313,49.023,159.483
C08718=1022.120,295.903,365.921,170.318,49.020,159.483
C08719=1022.127,296.150,365.889,170.322,49.017,159.483
C08720=1022.133,296.398,365.857,170.328,49.014,159.483
C08721=1022.139,296.646,365.824,170.332,49.011,159.483
C08722=1022.146,296.894,365.793,170.338,49.009,159.483
C08723=1022.152,297.141,365.760,170.342,49.006,159.483
C08724=1022.159,297.389,365.728,170.348,49.003,159.484
C08725=1022.165,297.637,365.696,170.354,49.001,159.484
C08726=1022.171,297.885,365.664,170.358,48.998,159.484
C08727=1022.178,298.132,365.631,170.364,48.996,159.484
C08728=1022.184,298.380,365.599,170.368,48.993,159.484
C08729=1022.191,298.628,365.567,170.374,48.990,159.485
C08730=1022.197,298.876,365.535,170.378,48.987,159.485
C08731=1022.203,299.124,365.502,170.384,48.985,159.485
C08732=1022.210,299.371,365.470,170.389,48.983,159.485
C08733=1022.217,299.619,365.437,170.394,48.979,159.485
C08734=1022.224,299.867,365.406,170.400,48.977,159.485
C08735=1022.230,300.115,365.373,170.404,48.975,159.486
C08736=1022.237,300.362,365.340,170.410,48.971,159.486
C08737=1022.243,300.610,365.309,170.414,48.969,159.486
C08738=1022.250,300.858,365.276,170.420,48.967,159.486
C08739=1022.257,301.106,365.244,170.425,48.964,159.486
C08740=1022.264,301.353,365.211,170.430,48.961,159.486
C08741=1022.270,301.602,365.179,170.436,48.959,159.487
C08742=1022.277,301.849,365.147,170.440,48.957,159.487
C08743=1022.283,302.097,365.114,170.446,48.953,159.487
C08744=1022.290,302.345,365.081,170.451,48.951,159.487
C08745=1022.297,302.592,365.049,170.456,48.949,159.487
C08746=1022.303,302.840,365.016,170.462,48.946,159.488
C08747=1022.310,303.088,364.985,170.466,48.943,159.488
C08748=1022.317,303.336,364.951,170.472,48.941,159.488
C08749=1022.323,303.584,364.919,170.478,48.938,159.488
C08750=1022.330,303.831,364.887,170.482,48.936,159.489
C08751=1022.337,304.079,364.853,170.488,48.934,159.489
C08752=1022.344,304.326,364.821,170.494,48.931,159.489
C08753=1022.350,304.574,364.789,170.498,48.929,159.489
C08754=1022.357,304.822,364.755,170.504,48.926,159.489
C08755=1022.364,305.070,364.723,170.509,48.923,159.490
C08756=1022.371,305.317,364.691,170.514,48.921,159.490
C08757=1022.377,305.565,364.657,170.520,48.918,159.490
C08758=1022.384,305.813,364.625,170.525,48.916,159.490
C08759=1022.391,306.060,364.593,170.530,48.914,159.491
C08760=1022.398,306.308,364.560,170.536,48.911,159.491
C08761=1022.405,306.556,364.527,170.541,48.909,159.491
C08762=1022.411,306.789,364.496,170.546,48.906,159.491
C08763=1022.418,307.022,364.466,170.551,48.904,159.491
C08764=1022.424,307.254,364.435,170.556,48.902,159.492
C08765=1022.430,307.487,364.404,170.561,48.899,159.492
C08766=1022.437,307.719,364.373,170.566,48.897,159.492
C08767=1022.444,307.952,364.342,170.571,48.895,159.492
C08768=1022.450,308.184,364.311,170.577,48.893,159.493
C08769=1022.457,308.417,364.280,170.581,48.891,159.493
C08770=1022.463,308.665,364.247,170.587,48.888,159.493
C08771=1022.471,308.912,364.215,170.593,48.886,159.494
C08772=1022.477,309.161,364.182,170.597,48.884,159.494
C08773=1022.484,309.407,364.149,170.603,48.881,159.494
C08774=1022.492,309.655,364.116,170.609,48.879,159.494
C08775=1022.498,309.903,364.083,170.613,48.876,159.494
C08776=1022.506,310.150,364.050,170.619,48.875,159.495
C08777=1022.512,310.398,364.017,170.625,48.872,159.495
C08778=1022.519,310.646,363.983,170.630,48.870,159.495
C08779=1022.525,310.894,363.950,170.636,48.868,159.496
C08780=1022.532,311.141,363.916,170.642,48.865,159.496
C08781=1022.539,311.388,363.883,170.647,48.864,159.497
C08782=1022.545,311.637,363.849,170.652,48.861,159.497
C08783=1022.551,311.884,363.816,170.657,48.859,159.497
C08784=1022.559,312.131,363.782,170.663,48.857,159.497
C08785=1022.565,312.378,363.748,170.669,48.855,159.498
C08786=1022.571,312.627,363.715,170.674,48.853,159.498
C08787=1022.578,312.874,363.681,170.679,48.851,159.498
C08788=1022.585,313.122,363.647,170.685,48.849,159.499
C08789=1022.592,313.369,363.614,170.690,48.847,159.499
C08790=1022.598,313.617,363.580,170.696,48.845,159.499
C08791=1022.605,313.865,363.546,170.702,48.843,159.500
C08792=1022.612,314.112,363.513,170.707,48.841,159.500
C08793=1022.618,314.360,363.479,170.713,48.839,159.501
C08794=1022.625,314.608,363.445,170.719,48.836,159.501
C08795=1022.632,314.855,363.411,170.724,48.835,159.501
C08796=1022.639,315.102,363.377,170.730,48.833,159.502
C08797=1022.645,315.351,363.344,170.735,48.830,159.502
C08798=1022.652,315.598,363.310,170.740,48.829,159.502
C08799=1022.659,315.845,363.277,170.746,48.827,159.503
C08800=1022.666,316.093,363.243,170.752,48.824,159.503
C08801=1022.672,316.340,363.209,170.757,48.823,159.503
C08802=1022.679,316.588,363.175,170.763,48.821,159.504
C08803=1022.687,316.836,363.141,170.769,48.818,159.504
C08804=1022.693,317.084,363.107,170.774,48.817,159.505
C08805=1022.700,317.331,363.073,170.780,48.815,159.505
C08806=1022.707,317.578,363.039,170.786,48.813,159.506
C08807=1022.714,317.825,363.005,170.792,48.811,159.506
C08808=1022.721,318.073,362.970,170.797,48.809,159.506
C08809=1022.728,318.321,362.936,170.803,48.807,159.507
C08810=1022.735,318.568,362.903,170.809,48.805,159.507
C08811=1022.741,318.816,362.869,170.815,48.803,159.508
C08812=1022.748,319.064,362.835,170.820,48.802,159.508
C08813=1022.756,319.311,362.801,170.826,48.799,159.508
C08814=1022.762,319.559,362.766,170.832,48.797,159.509
C08815=1022.770,319.806,362.732,170.838,48.796,159.509
C08816=1022.777,320.054,362.698,170.843,48.794,159.509
C08817=1022.784,320.302,362.664,170.849,48.792,159.510
C08818=1022.790,320.548,362.630,170.855,48.790,159.510
C08819=1022.797,320.796,362.596,170.861,48.788,159.511
C08820=1022.804,321.044,362.562,170.866,48.787,159.511
C08821=1022.811,321.292,362.528,170.872,48.785,159.512
C08822=1022.819,321.527,362.495,170.878,48.783,159.512
C08823=1022.825,321.762,362.462,170.883,48.781,159.513
C08824=1022.831,321.997,362.429,170.889,48.780,159.513
C08825=1022.839,322.232,362.397,170.894,48.778,159.513
C08826=1022.845,322.468,362.365,170.900,48.776,159.514
C08827=1022.852,322.703,362.332,170.905,48.775,159.514
C08828=1022.859,322.938,362.299,170.911,48.773,159.515
C08829=1022.865,323.173,362.267,170.916,48.771,159.515
C08830=1022.872,323.421,362.233,170.922,48.769,159.515
C08831=1022.879,323.668,362.198,170.928,48.767,159.516
C08832=1022.887,323.916,362.163,170.934,48.766,159.516
C08833=1022.894,324.163,362.129,170.940,48.765,159.517
C08834=1022.901,324.411,362.094,170.946,48.763,159.517
C08835=1022.908,324.658,362.060,170.952,48.761,159.518
C08836=1022.916,324.905,362.025,170.958,48.759,159.518
C08837=1022.923,325.153,361.992,170.964,48.757,159.519
C08838=1022.930,325.400,361.956,170.970,48.756,159.519
C08839=1022.937,325.648,361.923,170.976,48.754,159.520
C08840=1022.945,325.896,361.888,170.981,48.752,159.520
C08841=1022.952,326.143,361.853,170.987,48.751,159.521
C08842=1022.959,326.391,361.819,170.994,48.749,159.521
C08843=1022.967,326.638,361.784,171.000,48.747,159.522
C08844=1022.973,326.885,361.749,171.006,48.746,159.522
C08845=1022.982,327.133,361.714,171.012,48.744,159.523
C08846=1022.988,327.380,361.679,171.017,48.743,159.523
C08847=1022.995,327.628,361.644,171.023,48.741,159.524
C08848=1023.002,327.875,361.609,171.029,48.740,159.524
C08849=1023.009,328.122,361.574,171.035,48.738,159.525
C08850=1023.017,328.370,361.539,171.042,48.737,159.526
C08851=1023.024,328.618,361.504,171.048,48.735,159.526
C08852=1023.030,328.865,361.469,171.053,48.734,159.527
C08853=1023.038,329.112,361.434,171.060,48.732,159.527
C08854=1023.045,329.359,361.399,171.066,48.731,159.528
C08855=1023.052,329.608,361.363,171.072,48.729,159.528
C08856=1023.059,329.855,361.328,171.078,48.728,159.529
C08857=1023.065,330.102,361.293,171.084,48.726,159.529
C08858=1023.074,330.350,361.258,171.091,48.725,159.530
C08859=1023.081,330.597,361.222,171.096,48.723,159.530
C08860=1023.087,330.844,361.187,171.102,48.722,159.531
C08861=1023.095,331.092,361.152,171.109,48.721,159.532
C08862=1023.102,331.339,361.117,171.115,48.720,159.532
C08863=1023.109,331.587,361.082,171.121,48.718,159.533
C08864=1023.117,331.834,361.046,171.127,48.717,159.533
C08865=1023.124,332.081,361.011,171.134,48.715,159.534
C08866=1023.131,332.329,360.975,171.140,48.714,159.535
C08867=1023.139,332.576,360.940,171.146,48.712,159.535
C08868=1023.145,332.823,360.905,171.152,48.711,159.536
C08869=1023.153,333.071,360.869,171.158,48.710,159.536
C08870=1023.160,333.318,360.833,171.164,48.709,159.537
C08871=1023.167,333.566,360.798,171.171,48.708,159.538
C08872=1023.174,333.813,360.762,171.177,48.706,159.538
C08873=1023.182,334.061,360.727,171.183,48.705,159.539
C08874=1023.189,334.308,360.691,171.190,48.704,159.540
C08875=1023.196,334.556,360.655,171.196,48.703,159.540
C08876=1023.203,334.803,360.619,171.203,48.701,159.541
C08877=1023.211,335.050,360.583,171.209,48.700,159.542
C08878=1023.218,335.297,360.548,171.215,48.699,159.542
C08879=1023.225,335.545,360.512,171.222,48.698,159.543
C08880=1023.232,335.792,360.476,171.227,48.697,159.543
C08881=1023.240,336.040,360.440,171.233,48.695,159.544
C08882=1023.246,336.273,360.407,171.240,48.694,159.545
C08883=1023.254,336.505,360.373,171.246,48.693,159.545
C08884=1023.260,336.738,360.338,171.252,48.692,159.546
C08885=1023.268,336.971,360.305,171.258,48.691,159.547
C08886=1023.274,337.204,360.271,171.263,48.690,159.547
C08887=1023.282,337.437,360.238,171.270,48.688,159.548
C08888=1023.288,337.669,360.203,171.276,48.687,159.548
C08889=1023.295,337.902,360.169,171.282,48.687,159.549
C08890=1023.302,338.150,360.133,171.288,48.686,159.550
C08891=1023.310,338.397,360.097,171.295,48.684,159.551
C08892=1023.317,338.645,360.062,171.301,48.683,159.551
C08893=1023.324,338.892,360.025,171.308,48.683,159.552
C08894=1023.332,339.139,359.989,171.314,48.681,159.553
C08895=1023.340,339.387,359.953,171.320,48.680,159.553
C08896=1023.347,339.634,359.917,171.327,48.679,159.554
C08897=1023.354,339.881,359.881,171.334,48.678,159.555
C08898=1023.362,340.128,359.844,171.340,48.677,159.555
C08899=1023.369,340.375,359.808,171.347,48.676,159.556
C08900=1023.376,340.622,359.771,171.353,48.675,159.557
C08901=1023.384,340.870,359.735,171.360,48.674,159.558
C08902=1023.391,341.118,359.698,171.366,48.673,159.558
C08903=1023.398,341.364,359.662,171.373,48.673,159.559
C08904=1023.406,341.611,359.626,171.379,48.671,159.560
C08905=1023.414,341.859,359.589,171.386,48.671,159.561
C08906=1023.421,342.106,359.553,171.393,48.669,159.561
C08907=1023.429,342.353,359.516,171.400,48.668,159.562
C08908=1023.436,342.601,359.479,171.407,48.668,159.563
C08909=1023.443,342.848,359.443,171.413,48.667,159.564
C08910=1023.451,343.095,359.406,171.420,48.666,159.565
C08911=1023.458,343.342,359.370,171.426,48.665,159.565
C08912=1023.465,343.590,359.333,171.433,48.664,159.566
C08913=1023.473,343.837,359.296,171.440,48.663,159.567
C08914=1023.481,344.084,359.260,171.446,48.663,159.568
C08915=1023.488,344.331,359.222,171.453,48.662,159.568
C08916=1023.496,344.579,359.186,171.459,48.661,159.569
C08917=1023.503,344.826,359.149,171.466,48.660,159.570
C08918=1023.511,345.073,359.112,171.473,48.660,159.571
C08919=1023.519,345.320,359.075,171.479,48.658,159.572
C08920=1023.525,345.566,359.038,171.487,48.657,159.572
C08921=1023.533,345.813,359.001,171.494,48.657,159.573
C08922=1023.540,346.061,358.964,171.500,48.656,159.574
C08923=1023.549,346.309,358.927,171.507,48.656,159.575
C08924=1023.557,346.555,358.890,171.514,48.655,159.576
C08925=1023.564,346.803,358.853,171.521,48.654,159.577
C08926=1023.572,347.050,358.817,171.527,48.654,159.577
C08927=1023.579,347.297,358.779,171.535,48.653,159.578
C08928=1023.587,347.544,358.742,171.542,48.652,159.579
C08929=1023.595,347.791,358.706,171.548,48.651,159.580
C08930=1023.602,348.038,358.668,171.555,48.651,159.581
C08931=1023.609,348.286,358.631,171.562,48.650,159.582
C08932=1023.617,348.532,358.594,171.569,48.650,159.583
C08933=1023.624,348.780,358.556,171.575,48.649,159.583
C08934=1023.632,349.026,358.519,171.583,48.648,159.584
C08935=1023.640,349.274,358.482,171.590,48.647,159.585
C08936=1023.647,349.521,358.444,171.597,48.647,159.586
C08937=1023.655,349.768,358.407,171.604,48.647,159.587
C08938=1023.663,350.015,358.369,171.610,48.646,159.588
C08939=1023.670,350.262,358.331,171.618,48.645,159.589
C08940=1023.678,350.509,358.294,171.625,48.645,159.590
C08941=1023.686,350.757,358.256,171.632,48.644,159.591
C08942=1023.693,350.988,358.221,171.639,48.644,159.591
C08943=1023.700,351.219,358.187,171.645,48.643,159.592
C08944=1023.707,351.450,358.151,171.651,48.643,159.593
C08945=1023.714,351.682,358.116,171.658,48.643,159.594
C08946=1023.722,351.913,358.081,171.665,48.642,159.595
C08947=1023.729,352.145,358.046,171.671,48.642,159.596
C08948=1023.736,352.376,358.010,171.678,48.641,159.597
C08949=1023.744,352.607,357.975,171.685,48.641,159.598
C08950=1023.752,352.855,357.937,171.692,48.640,159.598
C08951=1023.759,353.101,357.899,171.699,48.640,159.599
C08952=1023.767,353.348,357.862,171.706,48.640,159.600
C08953=1023.775,353.595,357.823,171.713,48.639,159.601
C08954=1023.783,353.843,357.786,171.721,48.639,159.602
C08955=1023.792,354.089,357.748,171.727,48.638,159.603
C08956=1023.799,354.337,357.710,171.735,48.638,159.604
C08957=1023.806,354.583,357.672,171.742,48.638,159.605
C08958=1023.814,354.831,357.634,171.749,48.637,159.606
C08959=1023.823,355.077,357.596,171.757,48.637,159.607
C08960=1023.831,355.324,357.558,171.764,48.637,159.608
C08961=1023.838,355.572,357.520,171.771,48.636,159.609
C08962=1023.846,355.819,357.482,171.779,48.636,159.610
C08963=1023.854,356.065,357.443,171.786,48.636,159.611
C08964=1023.861,356.312,357.405,171.793,48.636,159.612
C08965=1023.869,356.560,357.367,171.801,48.635,159.613
C08966=1023.877,356.806,357.330,171.808,48.635,159.614
C08967=1023.885,357.053,357.291,171.815,48.634,159.615
C08968=1023.894,357.300,357.252,171.823,48.634,159.616
C08969=1023.901,357.547,357.214,171.830,48.634,159.617
C08970=1023.909,357.794,357.176,171.837,48.634,159.618
C08971=1023.917,358.040,357.137,171.845,48.634,159.619
C08972=1023.925,358.288,357.099,171.852,48.634,159.620
C08973=1023.933,358.535,357.060,171.860,48.633,159.622
C08974=1023.941,358.781,357.022,171.867,48.633,159.623
C08975=1023.950,359.028,356.984,171.874,48.633,159.624
C08976=1023.957,359.275,356.946,171.883,48.633,159.625
C08977=1023.965,359.522,356.907,171.890,48.633,159.626
C08978=1023.973,359.769,356.868,171.898,48.633,159.627
C08979=1023.981,360.016,356.830,171.905,48.632,159.628
C08980=1023.989,360.262,356.791,171.912,48.632,159.629
C08981=1023.998,360.510,356.752,171.920,48.632,159.630
C08982=1024.005,360.757,356.713,171.927,48.632,159.631
C08983=1024.013,361.003,356.674,171.935,48.632,159.632
C08984=1024.021,361.250,356.635,171.942,48.632,159.633
C08985=1024.029,361.497,356.597,171.950,48.632,159.634
C08986=1024.037,361.743,356.558,171.958,48.632,159.636
C08987=1024.044,361.991,356.519,171.966,48.632,159.637
C08988=1024.053,362.237,356.479,171.973,48.632,159.638
C08989=1024.061,362.485,356.441,171.981,48.632,159.639
C08990=1024.070,362.731,356.401,171.988,48.632,159.640
C08991=1024.077,362.978,356.363,171.997,48.632,159.641
C08992=1024.085,363.225,356.323,172.004,48.633,159.643
C08993=1024.093,363.471,356.284,172.012,48.632,159.644
C08994=1024.101,363.719,356.245,172.019,48.633,159.645
C08995=1024.110,363.965,356.206,172.027,48.632,159.646
C08996=1024.118,364.212,356.167,172.035,48.633,159.647
C08997=1024.126,364.459,356.127,172.043,48.633,159.648
C08998=1024.134,364.706,356.088,172.050,48.633,159.650
C08999=1024.142,364.952,356.049,172.058,48.633,159.651
C09000=1024.150,365.198,356.010,172.066,48.633,159.652
C09001=1024.159,365.446,355.971,172.074,48.634,159.653
C09002=1024.168,365.738,355.924,172.084,48.633,159.655
C09003=1024.179,366.031,355.877,172.093,48.633,159.656
C09004=1024.188,366.323,355.831,172.103,48.634,159.657
C09005=1024.198,366.616,355.784,172.111,48.634,159.659
C09006=1024.206,366.862,355.744,172.120,48.634,159.660
C09007=1024.215,367.109,355.705,172.128,48.635,159.661
C09008=1024.223,367.355,355.666,172.136,48.635,159.663
C09009=1024.231,367.602,355.626,172.144,48.635,159.664
C09010=1024.239,367.849,355.587,172.152,48.635,159.665
C09011=1024.248,368.096,355.547,172.159,48.636,159.666
C09012=1024.257,368.343,355.508,172.168,48.636,159.668
C09013=1024.265,368.589,355.467,172.176,48.636,159.669
C09014=1024.273,368.836,355.428,172.184,48.637,159.670
C09015=1024.281,369.083,355.388,172.192,48.637,159.671
C09016=1024.290,369.328,355.348,172.200,48.637,159.673
C09017=1024.298,369.575,355.308,172.208,48.638,159.674
C09018=1024.307,369.823,355.268,172.216,48.638,159.675
C09019=1024.315,370.069,355.227,172.225,48.638,159.676
C09020=1024.323,370.316,355.188,172.232,48.639,159.678
C09021=1024.331,370.562,355.147,172.241,48.640,159.679
C09022=1024.340,370.808,355.108,172.249,48.640,159.681
C09023=1024.348,371.055,355.067,172.258,48.640,159.682
C09024=1024.356,371.302,355.027,172.265,48.641,159.683
C09025=1024.365,371.548,354.987,172.274,48.641,159.685
C09026=1024.373,371.795,354.946,172.282,48.642,159.686
C09027=1024.382,372.042,354.907,172.291,48.642,159.687
C09028=1024.390,372.288,354.866,172.299,48.643,159.689
C09029=1024.399,372.535,354.826,172.307,48.643,159.690
C09030=1024.407,372.782,354.786,172.316,48.644,159.691
C09031=1024.416,373.028,354.746,172.324,48.644,159.693
C09032=1024.424,373.275,354.705,172.333,48.645,159.694
C09033=1024.433,373.521,354.665,172.341,48.645,159.695
C09034=1024.442,373.768,354.624,172.349,48.646,159.697
C09035=1024.449,374.015,354.584,172.357,48.647,159.698
C09036=1024.459,374.261,354.543,172.366,48.647,159.700
C09037=1024.467,374.508,354.503,172.375,48.648,159.701
C09038=1024.475,374.719,354.468,172.382,48.648,159.702
C09039=1024.482,374.931,354.433,172.389,48.649,159.703
C09040=1024.489,375.143,354.398,172.397,48.649,159.705
C09041=1024.497,375.354,354.363,172.404,48.650,159.706
C09042=1024.505,375.566,354.329,172.412,48.650,159.707
C09043=1024.512,375.778,354.294,172.419,48.651,159.708
C09044=1024.520,375.989,354.259,172.426,48.651,159.710
C09045=1024.527,376.201,354.224,172.434,48.652,159.711
C09046=1024.536,376.448,354.183,172.443,48.653,159.712
C09047=1024.545,376.694,354.142,172.451,48.653,159.714
C09048=1024.553,376.941,354.101,172.459,48.655,159.715
C09049=1024.562,377.187,354.061,172.468,48.655,159.717
C09050=1024.570,377.433,354.019,172.477,48.656,159.718
C09051=1024.579,377.680,353.978,172.485,48.657,159.720
C09052=1024.587,377.926,353.937,172.494,48.658,159.721
C09053=1024.596,378.173,353.896,172.503,48.659,159.723
C09054=1024.605,378.419,353.854,172.512,48.659,159.724
C09055=1024.614,378.665,353.814,172.520,48.660,159.726
C09056=1024.623,378.912,353.772,172.529,48.661,159.727
C09057=1024.631,379.159,353.731,172.538,48.662,159.729
C09058=1024.640,379.404,353.690,172.547,48.663,159.730
C09059=1024.649,379.651,353.648,172.555,48.663,159.732
C09060=1024.657,379.898,353.607,172.565,48.665,159.734
C09061=1024.666,380.144,353.565,172.574,48.665,159.735
C09062=1024.675,380.389,353.525,172.583,48.666,159.737
C09063=1024.684,380.635,353.483,172.592,48.667,159.738
C09064=1024.692,380.880,353.441,172.601,48.668,159.740
C09065=1024.702,381.126,353.400,172.610,48.669,159.741
C09066=1024.710,381.372,353.359,172.618,48.670,159.743
C09067=1024.719,381.617,353.318,172.628,48.671,159.745
C09068=1024.728,381.862,353.276,172.636,48.672,159.746
C09069=1024.737,382.109,353.234,172.645,48.673,159.748
C09070=1024.746,382.355,353.193,172.654,48.674,159.749
C09071=1024.755,382.601,353.151,172.664,48.675,159.751
C09072=1024.764,382.847,353.110,172.673,48.676,159.753
C09073=1024.773,383.094,353.068,172.682,48.677,159.754
C09074=1024.782,383.340,353.026,172.691,48.678,159.756
C09075=1024.791,383.586,352.985,172.700,48.680,159.757
C09076=1024.800,383.832,352.942,172.710,48.680,159.759
C09077=1024.809,384.079,352.900,172.719,48.681,159.761
C09078=1024.818,384.325,352.859,172.728,48.683,159.762
C09079=1024.827,384.571,352.817,172.738,48.684,159.764
C09080=1024.837,384.817,352.775,172.747,48.685,159.766
C09081=1024.846,385.063,352.733,172.756,48.686,159.767
C09082=1024.856,385.310,352.691,172.765,48.687,159.769
C09083=1024.865,385.556,352.649,172.775,48.688,159.771
C09084=1024.874,385.802,352.607,172.784,48.690,159.773
C09085=1024.883,386.049,352.565,172.793,48.691,159.774
C09086=1024.892,386.294,352.523,172.803,48.692,159.776
C09087=1024.902,386.541,352.480,172.812,48.693,159.778
C09088=1024.911,386.787,352.439,172.822,48.695,159.780
C09089=1024.919,387.033,352.395,172.832,48.696,159.781
C09090=1024.929,387.279,352.353,172.841,48.697,159.783
C09091=1024.938,387.526,352.311,172.851,48.698,159.785
C09092=1024.947,387.772,352.269,172.860,48.700,159.786
C09093=1024.957,388.018,352.226,172.869,48.701,159.788
C09094=1024.966,388.264,352.183,172.880,48.702,159.790
C09095=1024.975,388.510,352.140,172.889,48.704,159.792
C09096=1024.984,388.756,352.098,172.899,48.705,159.794
C09097=1024.994,389.002,352.055,172.908,48.706,159.795
C09098=1025.003,389.248,352.013,172.919,48.708,159.797
C09099=1025.012,389.495,351.969,172.928,48.709,159.799
C09100=1025.022,389.740,351.927,172.938,48.710,159.801
